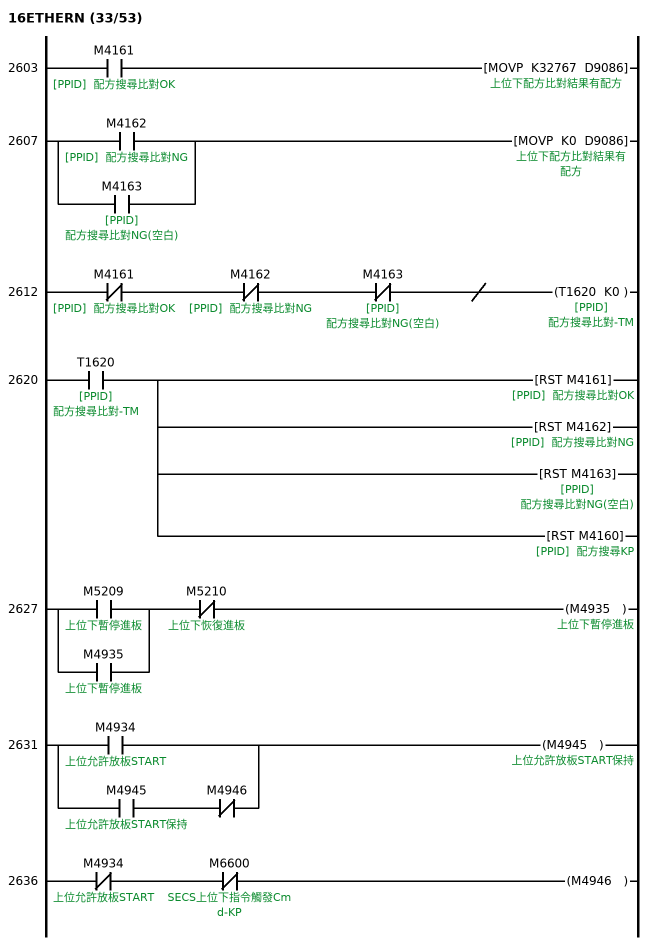
[picture p120: ladder of 16ETHERN, rungs at steps 2603 to 2636]
2603  LD      M4161  ; [PPID]  配方搜尋比對OK
      MOVP    K32767 D9086
2607  LD      M4162  ; [PPID]  配方搜尋比對NG
      OR      M4163  ; [PPID]  配方搜尋比對NG(空白)
      MOVP    K0 D9086
2612  LDI     M4161  ; [PPID]  配方搜尋比對OK
      ANI     M4162  ; [PPID]  配方搜尋比對NG
      ANI     M4163  ; [PPID]  配方搜尋比對NG(空白)
      INV
      OUT     T1620 K0  ; [PPID]  配方搜尋比對-TM
2620  LD      T1620  ; [PPID]  配方搜尋比對-TM
      RST     M4161  ; [PPID]  配方搜尋比對OK
      RST     M4162  ; [PPID]  配方搜尋比對NG
      RST     M4163  ; [PPID]  配方搜尋比對NG(空白)
      RST     M4160  ; [PPID]  配方搜尋KP
2627  LD      M5209  ; 上位下暫停進板
      OR      M4935  ; 上位下暫停進板
      ANI     M5210  ; 上位下恢復進板
      OUT     M4935  ; 上位下暫停進板
2631  LD      M4934  ; 上位允許放板START
      LD      M4945  ; 上位允許放板START保持
      ANI     M4946
      ORB
      OUT     M4945  ; 上位允許放板START保持
2636  LDI     M4934  ; 上位允許放板START
      ANI     M6600  ; SECS上位下指令觸發Cmd-KP
      OUT     M4946
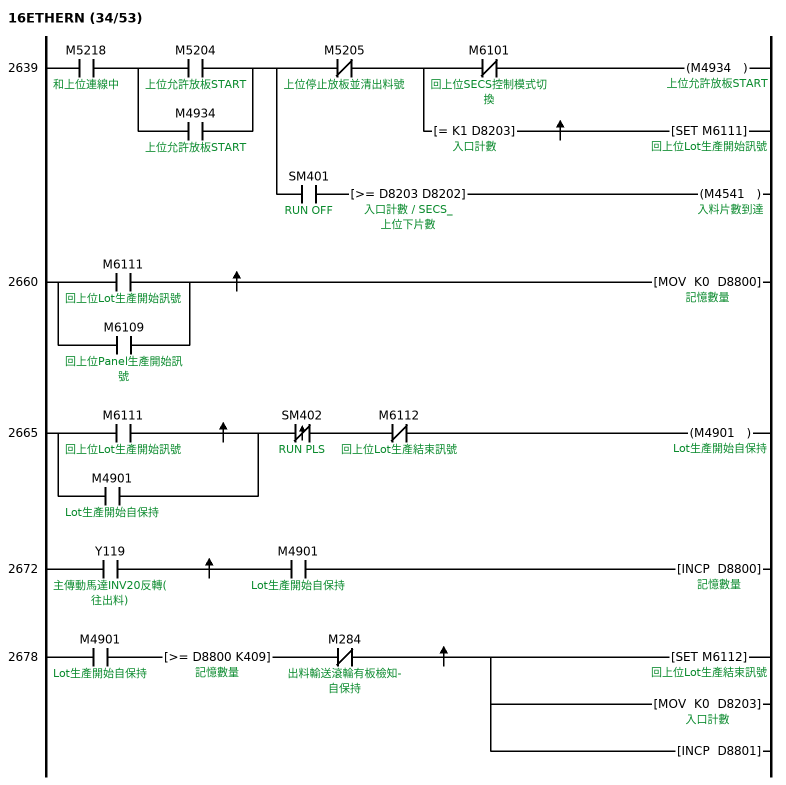
2639  LD      M5218  ; 和上位連線中
      LD      M5204  ; 上位允許放板START
      OR      M4934  ; 上位允許放板START
      ANB
      MPS
      ANI     M5205  ; 上位停止放板並清出料號
      MPS
      ANI     M6101  ; 回上位SECS控制模式切換
      OUT     M4934  ; 上位允許放板START
      MPP
      AND=    K1 D8203  ; 入口計數
      MEP
      SET     M6111  ; 回上位Lot生產開始訊號
      MPP
      AND     SM401  ; RUN OFF
      AND>=   D8203 D8202  ; 入口計數 / SECS_上位下片數
      OUT     M4541  ; 入料片數到達
2660  LD      M6111  ; 回上位Lot生產開始訊號
      OR      M6109  ; 回上位Panel生產開始訊號
      MEP
      MOV     K0 D8800  ; 記憶數量
2665  LD      M6111  ; 回上位Lot生產開始訊號
      MEP
      OR      M4901  ; Lot生產開始自保持
      ANDPI   SM402  ; RUN PLS
      ANI     M6112  ; 回上位Lot生產結束訊號
      OUT     M4901  ; Lot生產開始自保持
2672  LD      Y119  ; 主傳動馬達INV20反轉(往出料)
      MEP
      AND     M4901  ; Lot生產開始自保持
      INCP    D8800
2678  LD      M4901  ; Lot生產開始自保持
      AND>=   D8800 K409  ; 記憶數量
      ANI     M284  ; 出料輸送滾輪有板檢知-自保持
      MEP
      SET     M6112  ; 回上位Lot生產結束訊號
      MOV     K0 D8203
      INCP    D8801
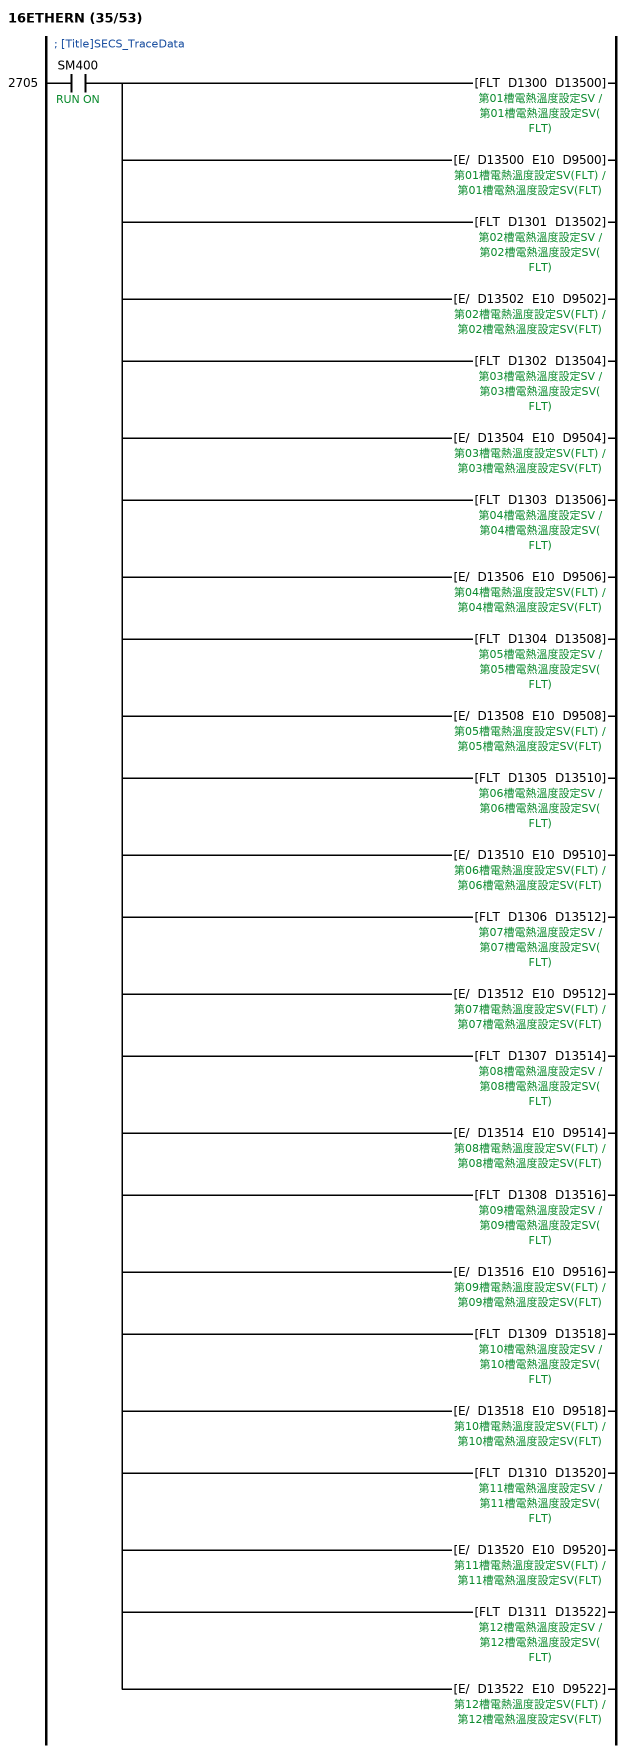
; [Title]SECS_TraceData
2705  LD      SM400  ; RUN ON
      FLT     D1300 D13500  ; 第01槽電熱溫度設定SV / 第01槽電熱溫度設定SV(FLT)
      E/      D13500 E10 D9500  ; 第01槽電熱溫度設定SV(FLT)
      FLT     D1301 D13502  ; 第02槽電熱溫度設定SV / 第02槽電熱溫度設定SV(FLT)
      E/      D13502 E10 D9502  ; 第02槽電熱溫度設定SV(FLT)
      FLT     D1302 D13504  ; 第03槽電熱溫度設定SV / 第03槽電熱溫度設定SV(FLT)
      E/      D13504 E10 D9504  ; 第03槽電熱溫度設定SV(FLT)
      FLT     D1303 D13506  ; 第04槽電熱溫度設定SV / 第04槽電熱溫度設定SV(FLT)
      E/      D13506 E10 D9506  ; 第04槽電熱溫度設定SV(FLT)
      FLT     D1304 D13508  ; 第05槽電熱溫度設定SV / 第05槽電熱溫度設定SV(FLT)
      E/      D13508 E10 D9508  ; 第05槽電熱溫度設定SV(FLT)
      FLT     D1305 D13510  ; 第06槽電熱溫度設定SV / 第06槽電熱溫度設定SV(FLT)
      E/      D13510 E10 D9510  ; 第06槽電熱溫度設定SV(FLT)
      FLT     D1306 D13512  ; 第07槽電熱溫度設定SV / 第07槽電熱溫度設定SV(FLT)
      E/      D13512 E10 D9512  ; 第07槽電熱溫度設定SV(FLT)
      FLT     D1307 D13514  ; 第08槽電熱溫度設定SV / 第08槽電熱溫度設定SV(FLT)
      E/      D13514 E10 D9514  ; 第08槽電熱溫度設定SV(FLT)
      FLT     D1308 D13516  ; 第09槽電熱溫度設定SV / 第09槽電熱溫度設定SV(FLT)
      E/      D13516 E10 D9516  ; 第09槽電熱溫度設定SV(FLT)
      FLT     D1309 D13518  ; 第10槽電熱溫度設定SV / 第10槽電熱溫度設定SV(FLT)
      E/      D13518 E10 D9518  ; 第10槽電熱溫度設定SV(FLT)
      FLT     D1310 D13520  ; 第11槽電熱溫度設定SV / 第11槽電熱溫度設定SV(FLT)
      E/      D13520 E10 D9520  ; 第11槽電熱溫度設定SV(FLT)
      FLT     D1311 D13522  ; 第12槽電熱溫度設定SV / 第12槽電熱溫度設定SV(FLT)
      E/      D13522 E10 D9522  ; 第12槽電熱溫度設定SV(FLT)
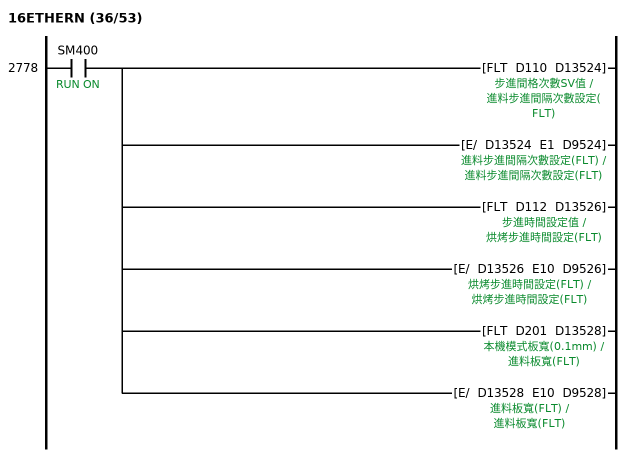
2778  LD      SM400  ; RUN ON
      FLT     D110 D13524  ; 步進間格次數SV值 / 進料步進間隔次數設定(FLT)
      E/      D13524 E1 D9524  ; 進料步進間隔次數設定(FLT)
      FLT     D112 D13526  ; 步進時間設定值 / 烘烤步進時間設定(FLT)
      E/      D13526 E10 D9526  ; 烘烤步進時間設定(FLT)
      FLT     D201 D13528  ; 進料板寬(FLT)
      E/      D13528 E10 D9528  ; 進料板寬(FLT)
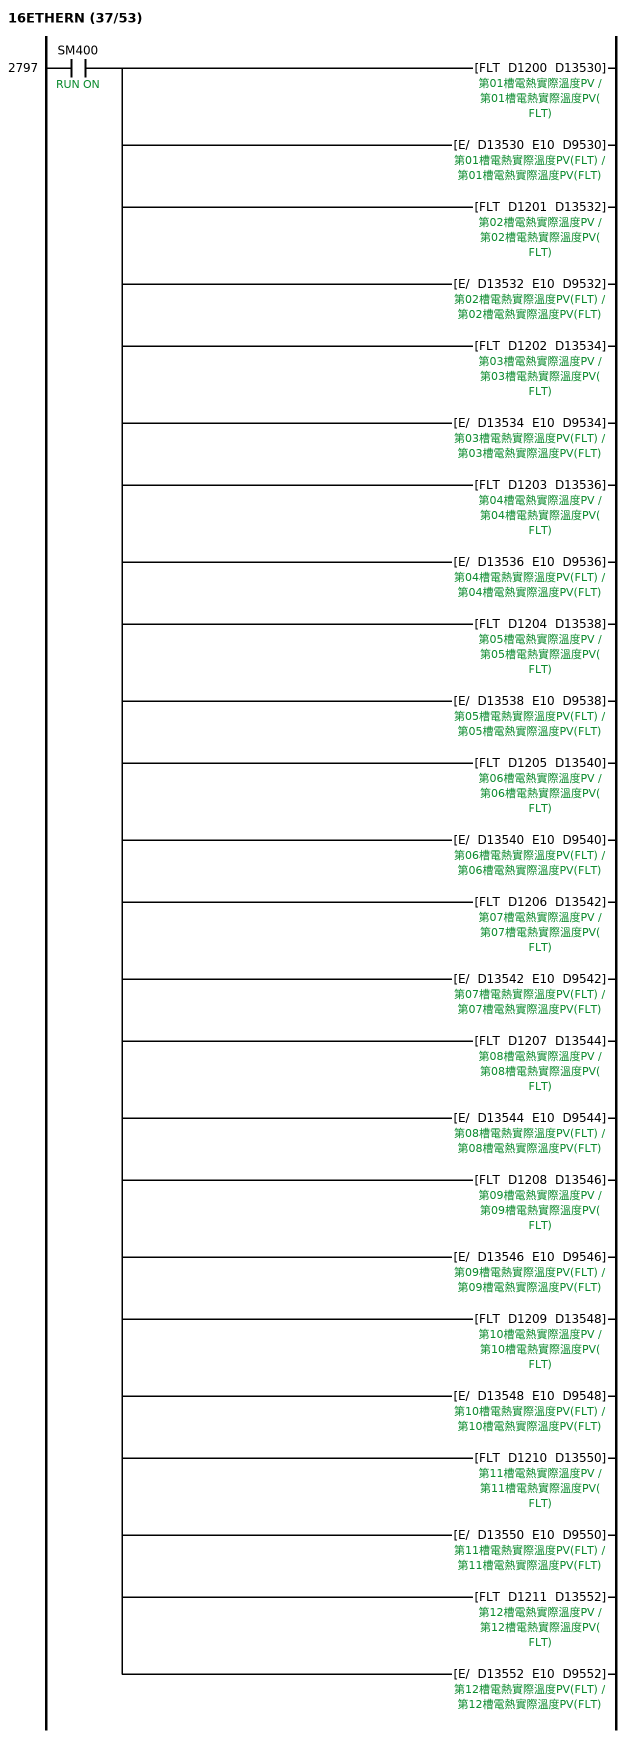
2797  LD      SM400  ; RUN ON
      FLT     D1200 D13530  ; 第01槽電熱實際溫度PV(FLT)
      E/      D13530 E10 D9530  ; 第01槽電熱實際溫度PV(FLT)
      FLT     D1201 D13532  ; 第02槽電熱實際溫度PV(FLT)
      E/      D13532 E10 D9532  ; 第02槽電熱實際溫度PV(FLT)
      FLT     D1202 D13534  ; 第03槽電熱實際溫度PV(FLT)
      E/      D13534 E10 D9534  ; 第03槽電熱實際溫度PV(FLT)
      FLT     D1203 D13536  ; 第04槽電熱實際溫度PV(FLT)
      E/      D13536 E10 D9536  ; 第04槽電熱實際溫度PV(FLT)
      FLT     D1204 D13538  ; 第05槽電熱實際溫度PV(FLT)
      E/      D13538 E10 D9538  ; 第05槽電熱實際溫度PV(FLT)
      FLT     D1205 D13540  ; 第06槽電熱實際溫度PV(FLT)
      E/      D13540 E10 D9540  ; 第06槽電熱實際溫度PV(FLT)
      FLT     D1206 D13542  ; 第07槽電熱實際溫度PV(FLT)
      E/      D13542 E10 D9542  ; 第07槽電熱實際溫度PV(FLT)
      FLT     D1207 D13544  ; 第08槽電熱實際溫度PV(FLT)
      E/      D13544 E10 D9544  ; 第08槽電熱實際溫度PV(FLT)
      FLT     D1208 D13546  ; 第09槽電熱實際溫度PV(FLT)
      E/      D13546 E10 D9546  ; 第09槽電熱實際溫度PV(FLT)
      FLT     D1209 D13548  ; 第10槽電熱實際溫度PV(FLT)
      E/      D13548 E10 D9548  ; 第10槽電熱實際溫度PV(FLT)
      FLT     D1210 D13550  ; 第11槽電熱實際溫度PV(FLT)
      E/      D13550 E10 D9550  ; 第11槽電熱實際溫度PV(FLT)
      FLT     D1211 D13552  ; 第12槽電熱實際溫度PV(FLT)
      E/      D13552 E10 D9552  ; 第12槽電熱實際溫度PV(FLT)
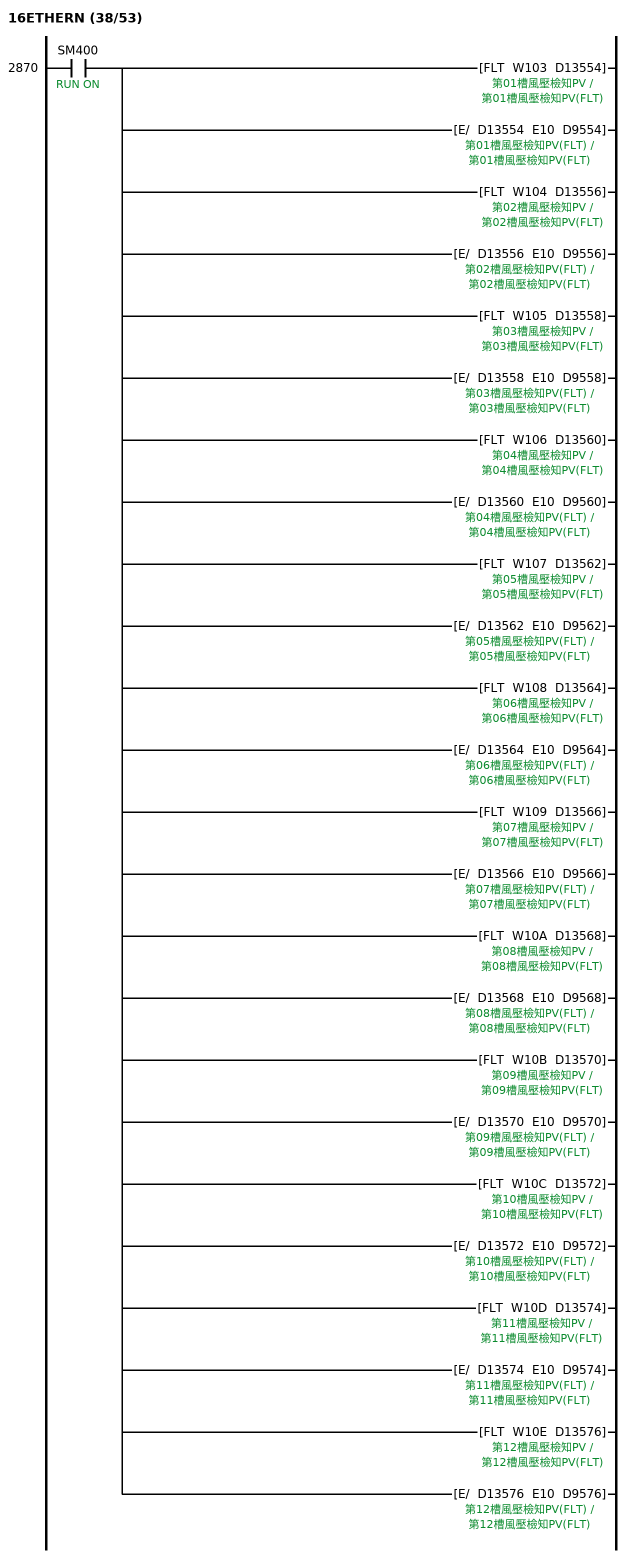
2870  LD      SM400  ; RUN ON
      FLT     W103 D13554  ; 第01槽風壓檢知PV / 第01槽風壓檢知PV(FLT)
      E/      D13554 E10 D9554  ; 第01槽風壓檢知PV(FLT)
      FLT     W104 D13556  ; 第02槽風壓檢知PV / 第02槽風壓檢知PV(FLT)
      E/      D13556 E10 D9556  ; 第02槽風壓檢知PV(FLT)
      FLT     W105 D13558  ; 第03槽風壓檢知PV / 第03槽風壓檢知PV(FLT)
      E/      D13558 E10 D9558  ; 第03槽風壓檢知PV(FLT)
      FLT     W106 D13560  ; 第04槽風壓檢知PV / 第04槽風壓檢知PV(FLT)
      E/      D13560 E10 D9560  ; 第04槽風壓檢知PV(FLT)
      FLT     W107 D13562  ; 第05槽風壓檢知PV / 第05槽風壓檢知PV(FLT)
      E/      D13562 E10 D9562  ; 第05槽風壓檢知PV(FLT)
      FLT     W108 D13564  ; 第06槽風壓檢知PV / 第06槽風壓檢知PV(FLT)
      E/      D13564 E10 D9564  ; 第06槽風壓檢知PV(FLT)
      FLT     W109 D13566  ; 第07槽風壓檢知PV / 第07槽風壓檢知PV(FLT)
      E/      D13566 E10 D9566  ; 第07槽風壓檢知PV(FLT)
      FLT     W10A D13568  ; 第08槽風壓檢知PV / 第08槽風壓檢知PV(FLT)
      E/      D13568 E10 D9568  ; 第08槽風壓檢知PV(FLT)
      FLT     W10B D13570  ; 第09槽風壓檢知PV / 第09槽風壓檢知PV(FLT)
      E/      D13570 E10 D9570  ; 第09槽風壓檢知PV(FLT)
      FLT     W10C D13572  ; 第10槽風壓檢知PV / 第10槽風壓檢知PV(FLT)
      E/      D13572 E10 D9572  ; 第10槽風壓檢知PV(FLT)
      FLT     W10D D13574  ; 第11槽風壓檢知PV / 第11槽風壓檢知PV(FLT)
      E/      D13574 E10 D9574  ; 第11槽風壓檢知PV(FLT)
      FLT     W10E D13576  ; 第12槽風壓檢知PV / 第12槽風壓檢知PV(FLT)
      E/      D13576 E10 D9576  ; 第12槽風壓檢知PV(FLT)
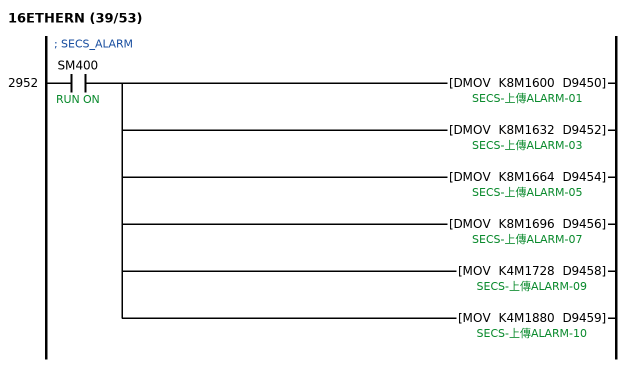
; SECS_ALARM
2952  LD      SM400  ; RUN ON
      DMOV    K8M1600 D9450  ; SECS-上傳ALARM-01
      DMOV    K8M1632 D9452  ; SECS-上傳ALARM-03
      DMOV    K8M1664 D9454  ; 出料風車1過載異常 / SECS-上傳ALARM-05
      DMOV    K8M1696 D9456  ; 進料夾爪開異常 / SECS-上傳ALARM-07
      MOV     K4M1728 D9458  ; 緊急停止異常 / SECS-上傳ALARM-09
      MOV     K4M1880 D9459  ; #01分路開關跳脫 / SECS-上傳ALARM-10
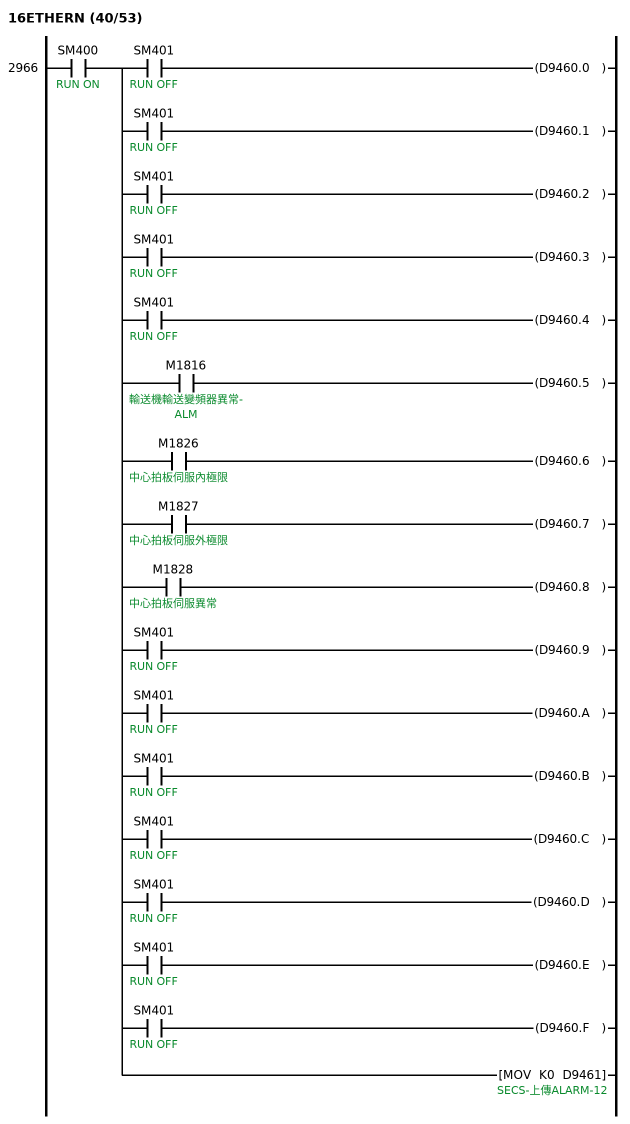
2966  LD      SM400  ; RUN ON
      MPS
      AND     SM401  ; RUN OFF
      OUT     D9460.0
      MRD
      AND     SM401  ; RUN OFF
      OUT     D9460.1
      MRD
      AND     SM401  ; RUN OFF
      OUT     D9460.2
      MRD
      AND     SM401  ; RUN OFF
      OUT     D9460.3
      MRD
      AND     SM401  ; RUN OFF
      OUT     D9460.4
      MRD
      AND     M1816  ; 輸送機輸送變頻器異常-ALM
      OUT     D9460.5
      MRD
      AND     M1826  ; 中心拍板伺服內極限
      OUT     D9460.6
      MRD
      AND     M1827  ; 中心拍板伺服外極限
      OUT     D9460.7
      MRD
      AND     M1828  ; 中心拍板伺服異常
      OUT     D9460.8
      MRD
      AND     SM401  ; RUN OFF
      OUT     D9460.9
      MRD
      AND     SM401  ; RUN OFF
      OUT     D9460.A
      MRD
      AND     SM401  ; RUN OFF
      OUT     D9460.B
      MRD
      AND     SM401  ; RUN OFF
      OUT     D9460.C
      MRD
      AND     SM401  ; RUN OFF
      OUT     D9460.D
      MRD
      AND     SM401  ; RUN OFF
      OUT     D9460.E
      MRD
      AND     SM401  ; RUN OFF
      OUT     D9460.F
      MPP
      MOV     K0 D9461  ; SECS-上傳ALARM-12
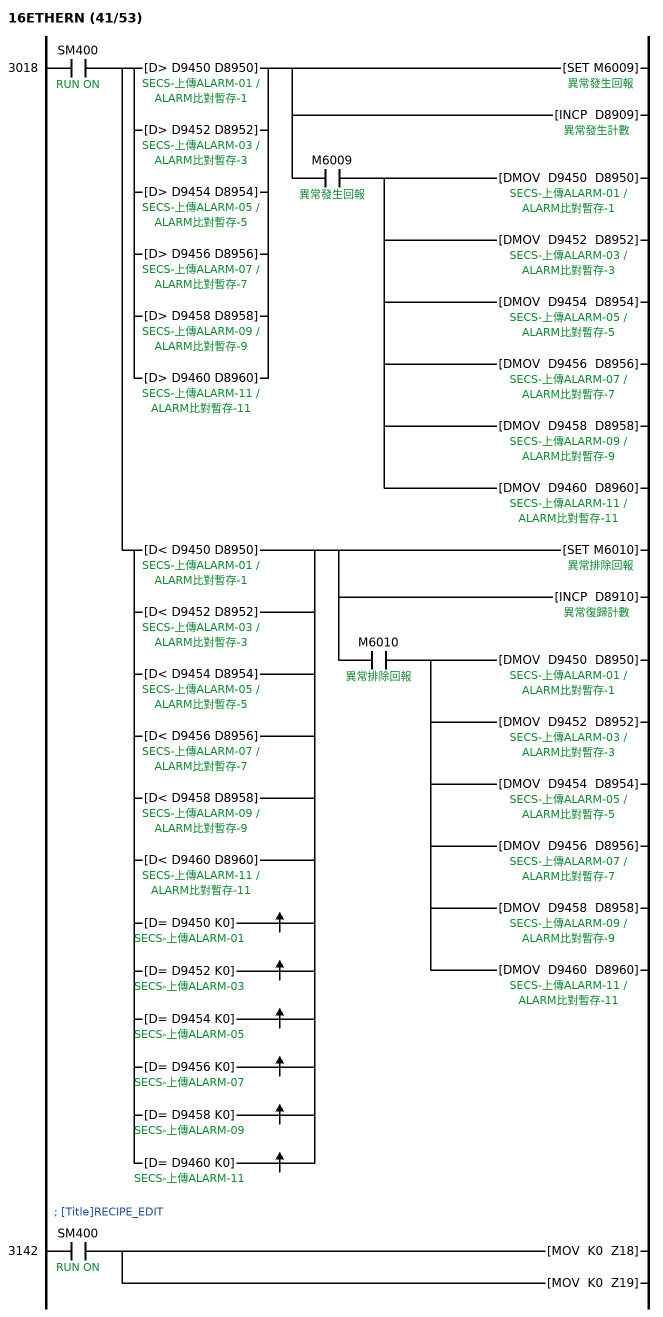
3018  LD      SM400  ; RUN ON
      MPS
      LDD>    D9450 D8950  ; SECS-上傳ALARM-01 / ALARM比對暫存-1
      ORD>    D9452 D8952  ; SECS-上傳ALARM-03 / ALARM比對暫存-3
      ORD>    D9454 D8954  ; SECS-上傳ALARM-05 / ALARM比對暫存-5
      ORD>    D9456 D8956  ; SECS-上傳ALARM-07 / ALARM比對暫存-7
      ORD>    D9458 D8958  ; SECS-上傳ALARM-09 / ALARM比對暫存-9
      ORD>    D9460 D8960  ; SECS-上傳ALARM-11 / ALARM比對暫存-11
      ANB
      SET     M6009  ; 異常發生回報
      INCP    D8909  ; 異常發生計數
      AND     M6009  ; 異常發生回報
      DMOV    D9450 D8950
      DMOV    D9452 D8952
      DMOV    D9454 D8954
      DMOV    D9456 D8956
      DMOV    D9458 D8958
      DMOV    D9460 D8960
      MPP
      LDD<    D9450 D8950  ; SECS-上傳ALARM-01 / ALARM比對暫存-1
      ORD<    D9452 D8952  ; SECS-上傳ALARM-03 / ALARM比對暫存-3
      ORD<    D9454 D8954  ; SECS-上傳ALARM-05 / ALARM比對暫存-5
      ORD<    D9456 D8956  ; SECS-上傳ALARM-07 / ALARM比對暫存-7
      ORD<    D9458 D8958  ; SECS-上傳ALARM-09 / ALARM比對暫存-9
      ORD<    D9460 D8960  ; SECS-上傳ALARM-11 / ALARM比對暫存-11
      LDD=    D9450 K0  ; SECS-上傳ALARM-01
      MEP
      ORB
      LDD=    D9452 K0  ; SECS-上傳ALARM-03
      MEP
      ORB
      LDD=    D9454 K0  ; SECS-上傳ALARM-05
      MEP
      ORB
      LDD=    D9456 K0  ; SECS-上傳ALARM-07
      MEP
      ORB
      LDD=    D9458 K0  ; SECS-上傳ALARM-09
      MEP
      ORB
      LDD=    D9460 K0  ; SECS-上傳ALARM-11
      MEP
      ORB
      ANB
      SET     M6010  ; 異常排除回報
      INCP    D8910  ; 異常復歸計數
      AND     M6010  ; 異常排除回報
      DMOV    D9450 D8950
      DMOV    D9452 D8952
      DMOV    D9454 D8954
      DMOV    D9456 D8956
      DMOV    D9458 D8958
      DMOV    D9460 D8960
; [Title]RECIPE_EDIT
3142  LD      SM400  ; RUN ON
      MOV     K0 Z18
      MOV     K0 Z19
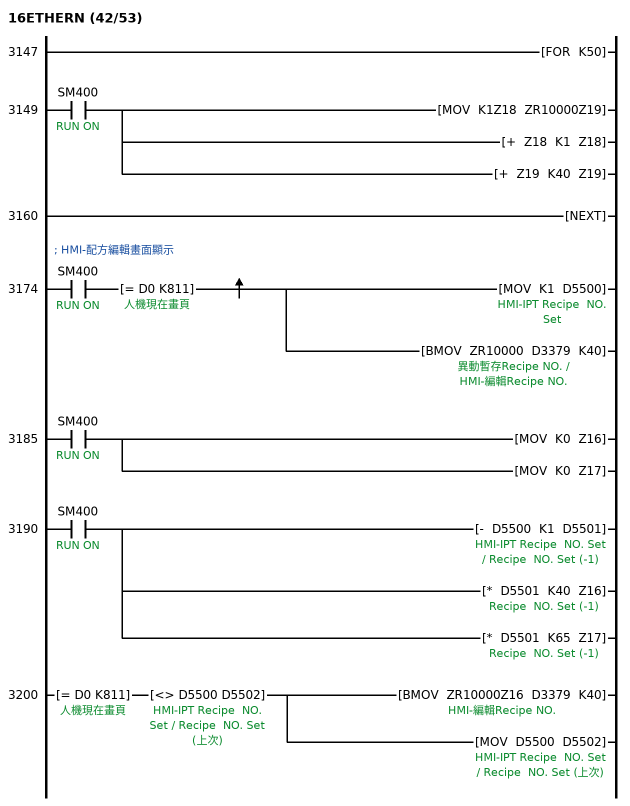
3147  FOR     K50
3149  LD      SM400  ; RUN ON
      MOV     K1Z18 ZR10000Z19
      +       Z18 K1 Z18
      +       Z19 K40 Z19
3160  NEXT
; HMI-配方編輯畫面顯示
3174  LD      SM400  ; RUN ON
      AND=    D0 K811  ; 人機現在畫頁
      MEP
      MOV     K1 D5500  ; HMI-IPT Recipe  NO. Set
      BMOV    ZR10000 D3379 K40  ; 異動暫存Recipe NO. / HMI-編輯Recipe NO.
3185  LD      SM400  ; RUN ON
      MOV     K0 Z16
      MOV     K0 Z17
3190  LD      SM400  ; RUN ON
      -       D5500 K1 D5501  ; Recipe  NO. Set (-1)
      *       D5501 K40 Z16
      *       D5501 K65 Z17
3200  LD=     D0 K811  ; 人機現在畫頁
      AND<>   D5500 D5502  ; HMI-IPT Recipe  NO. Set / Recipe  NO. Set (上次)
      BMOV    ZR10000Z16 D3379 K40
      MOV     D5500 D5502
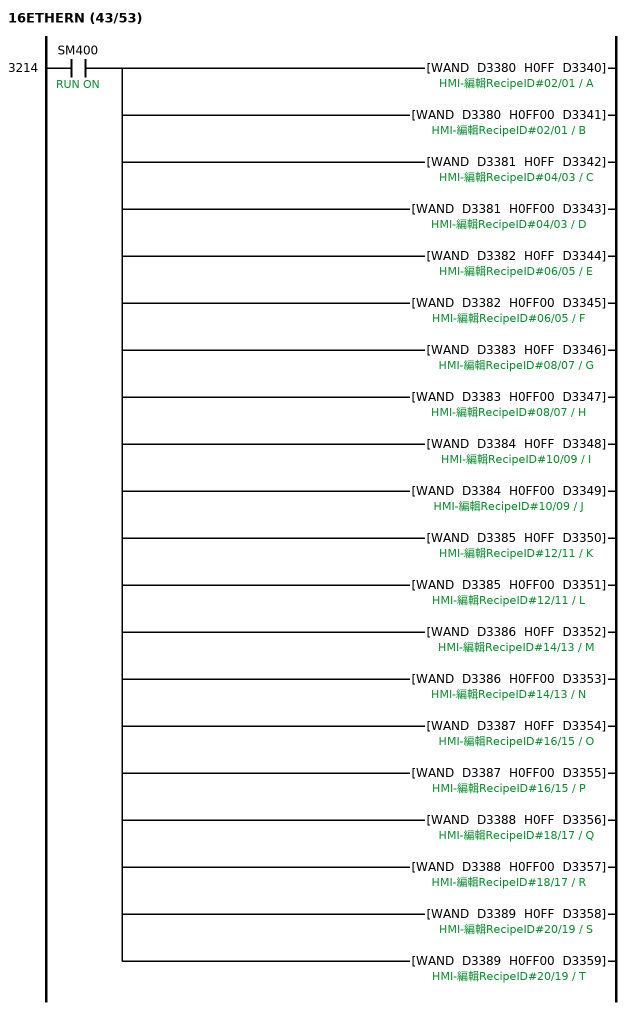
3214  LD      SM400  ; RUN ON
      WAND    D3380 H0FF D3340  ; HMI-編輯RecipeID#02/01 / A
      WAND    D3380 H0FF00 D3341  ; B
      WAND    D3381 H0FF D3342  ; HMI-編輯RecipeID#04/03 / C
      WAND    D3381 H0FF00 D3343  ; D
      WAND    D3382 H0FF D3344  ; HMI-編輯RecipeID#06/05 / E
      WAND    D3382 H0FF00 D3345  ; F
      WAND    D3383 H0FF D3346  ; HMI-編輯RecipeID#08/07 / G
      WAND    D3383 H0FF00 D3347  ; H
      WAND    D3384 H0FF D3348  ; HMI-編輯RecipeID#10/09 / I
      WAND    D3384 H0FF00 D3349  ; J
      WAND    D3385 H0FF D3350  ; HMI-編輯RecipeID#12/11 / K
      WAND    D3385 H0FF00 D3351  ; L
      WAND    D3386 H0FF D3352  ; HMI-編輯RecipeID#14/13 / M
      WAND    D3386 H0FF00 D3353  ; N
      WAND    D3387 H0FF D3354  ; HMI-編輯RecipeID#16/15 / O
      WAND    D3387 H0FF00 D3355  ; P
      WAND    D3388 H0FF D3356  ; HMI-編輯RecipeID#18/17 / Q
      WAND    D3388 H0FF00 D3357  ; R
      WAND    D3389 H0FF D3358  ; HMI-編輯RecipeID#20/19 / S
      WAND    D3389 H0FF00 D3359  ; T
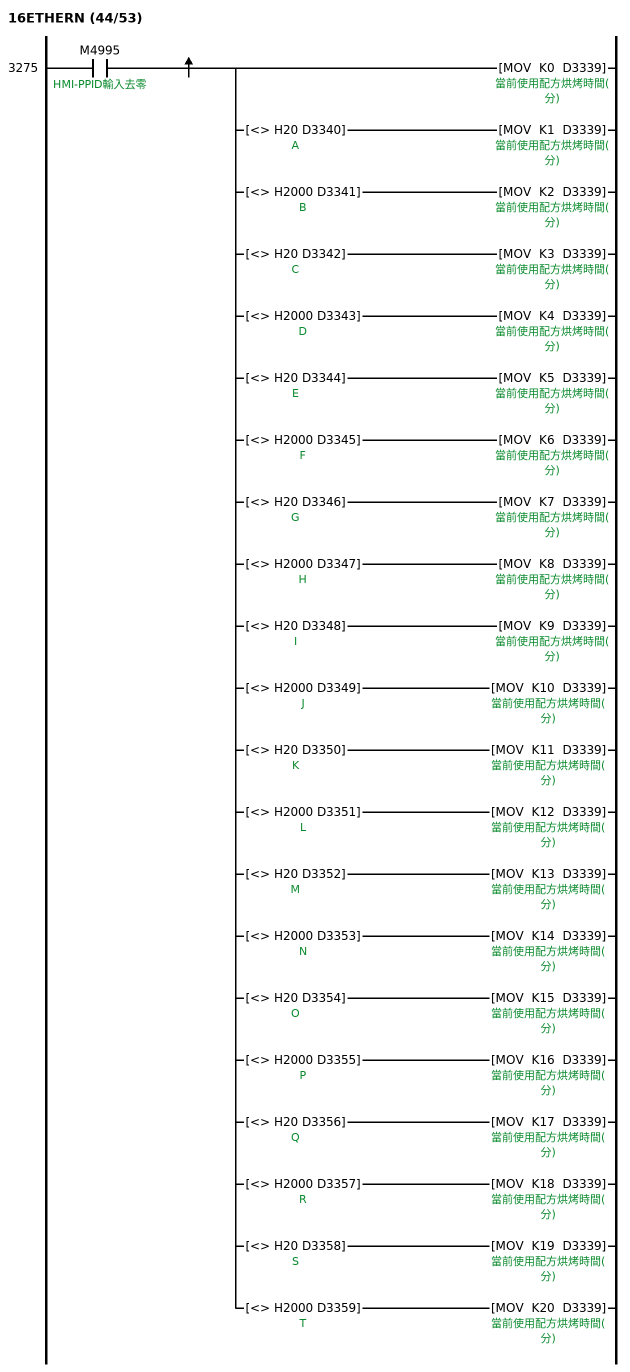
3275  LD      M4995  ; HMI-PPID輸入去零
      MEP
      MOV     K0 D3339  ; 當前使用配方烘烤時間(分)
      MPS
      AND<>   H20 D3340  ; A
      MOV     K1 D3339
      MRD
      AND<>   H2000 D3341  ; B
      MOV     K2 D3339
      MRD
      AND<>   H20 D3342  ; C
      MOV     K3 D3339
      MRD
      AND<>   H2000 D3343  ; D
      MOV     K4 D3339
      MRD
      AND<>   H20 D3344  ; E
      MOV     K5 D3339
      MRD
      AND<>   H2000 D3345  ; F
      MOV     K6 D3339
      MRD
      AND<>   H20 D3346  ; G
      MOV     K7 D3339
      MRD
      AND<>   H2000 D3347  ; H
      MOV     K8 D3339
      MRD
      AND<>   H20 D3348  ; I
      MOV     K9 D3339
      MRD
      AND<>   H2000 D3349  ; J
      MOV     K10 D3339
      MRD
      AND<>   H20 D3350  ; K
      MOV     K11 D3339
      MRD
      AND<>   H2000 D3351  ; L
      MOV     K12 D3339
      MRD
      AND<>   H20 D3352  ; M
      MOV     K13 D3339
      MRD
      AND<>   H2000 D3353  ; N
      MOV     K14 D3339
      MRD
      AND<>   H20 D3354  ; O
      MOV     K15 D3339
      MRD
      AND<>   H2000 D3355  ; P
      MOV     K16 D3339
      MRD
      AND<>   H20 D3356  ; Q
      MOV     K17 D3339
      MRD
      AND<>   H2000 D3357  ; R
      MOV     K18 D3339
      MRD
      AND<>   H20 D3358  ; S
      MOV     K19 D3339
      MPP
      AND<>   H2000 D3359  ; T
      MOV     K20 D3339
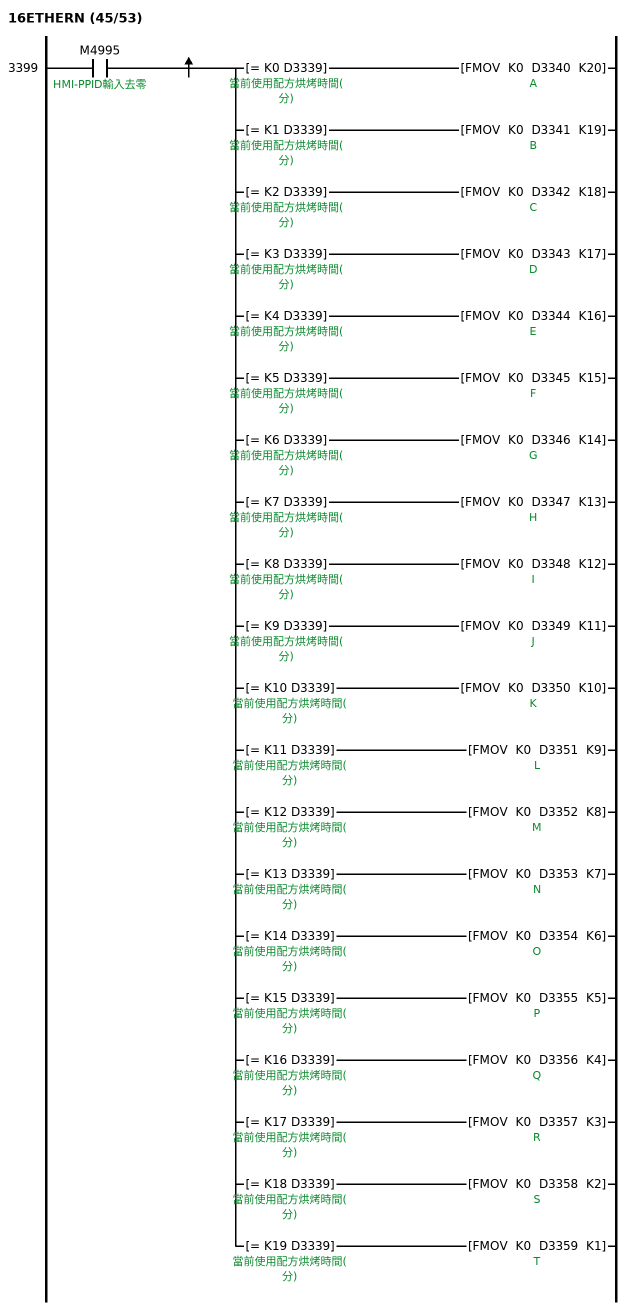
3399  LD      M4995  ; HMI-PPID輸入去零
      MEP
      MPS
      AND=    K0 D3339  ; 當前使用配方烘烤時間(分)
      FMOV    K0 D3340 K20
      MRD
      AND=    K1 D3339  ; 當前使用配方烘烤時間(分)
      FMOV    K0 D3341 K19
      MRD
      AND=    K2 D3339  ; 當前使用配方烘烤時間(分)
      FMOV    K0 D3342 K18
      MRD
      AND=    K3 D3339  ; 當前使用配方烘烤時間(分)
      FMOV    K0 D3343 K17
      MRD
      AND=    K4 D3339  ; 當前使用配方烘烤時間(分)
      FMOV    K0 D3344 K16
      MRD
      AND=    K5 D3339  ; 當前使用配方烘烤時間(分)
      FMOV    K0 D3345 K15
      MRD
      AND=    K6 D3339  ; 當前使用配方烘烤時間(分)
      FMOV    K0 D3346 K14
      MRD
      AND=    K7 D3339  ; 當前使用配方烘烤時間(分)
      FMOV    K0 D3347 K13
      MRD
      AND=    K8 D3339  ; 當前使用配方烘烤時間(分)
      FMOV    K0 D3348 K12
      MRD
      AND=    K9 D3339  ; 當前使用配方烘烤時間(分)
      FMOV    K0 D3349 K11
      MRD
      AND=    K10 D3339  ; 當前使用配方烘烤時間(分)
      FMOV    K0 D3350 K10
      MRD
      AND=    K11 D3339  ; 當前使用配方烘烤時間(分)
      FMOV    K0 D3351 K9
      MRD
      AND=    K12 D3339  ; 當前使用配方烘烤時間(分)
      FMOV    K0 D3352 K8
      MRD
      AND=    K13 D3339  ; 當前使用配方烘烤時間(分)
      FMOV    K0 D3353 K7
      MRD
      AND=    K14 D3339  ; 當前使用配方烘烤時間(分)
      FMOV    K0 D3354 K6
      MRD
      AND=    K15 D3339  ; 當前使用配方烘烤時間(分)
      FMOV    K0 D3355 K5
      MRD
      AND=    K16 D3339  ; 當前使用配方烘烤時間(分)
      FMOV    K0 D3356 K4
      MRD
      AND=    K17 D3339  ; 當前使用配方烘烤時間(分)
      FMOV    K0 D3357 K3
      MRD
      AND=    K18 D3339  ; 當前使用配方烘烤時間(分)
      FMOV    K0 D3358 K2
      MPP
      AND=    K19 D3339  ; 當前使用配方烘烤時間(分)
      FMOV    K0 D3359 K1
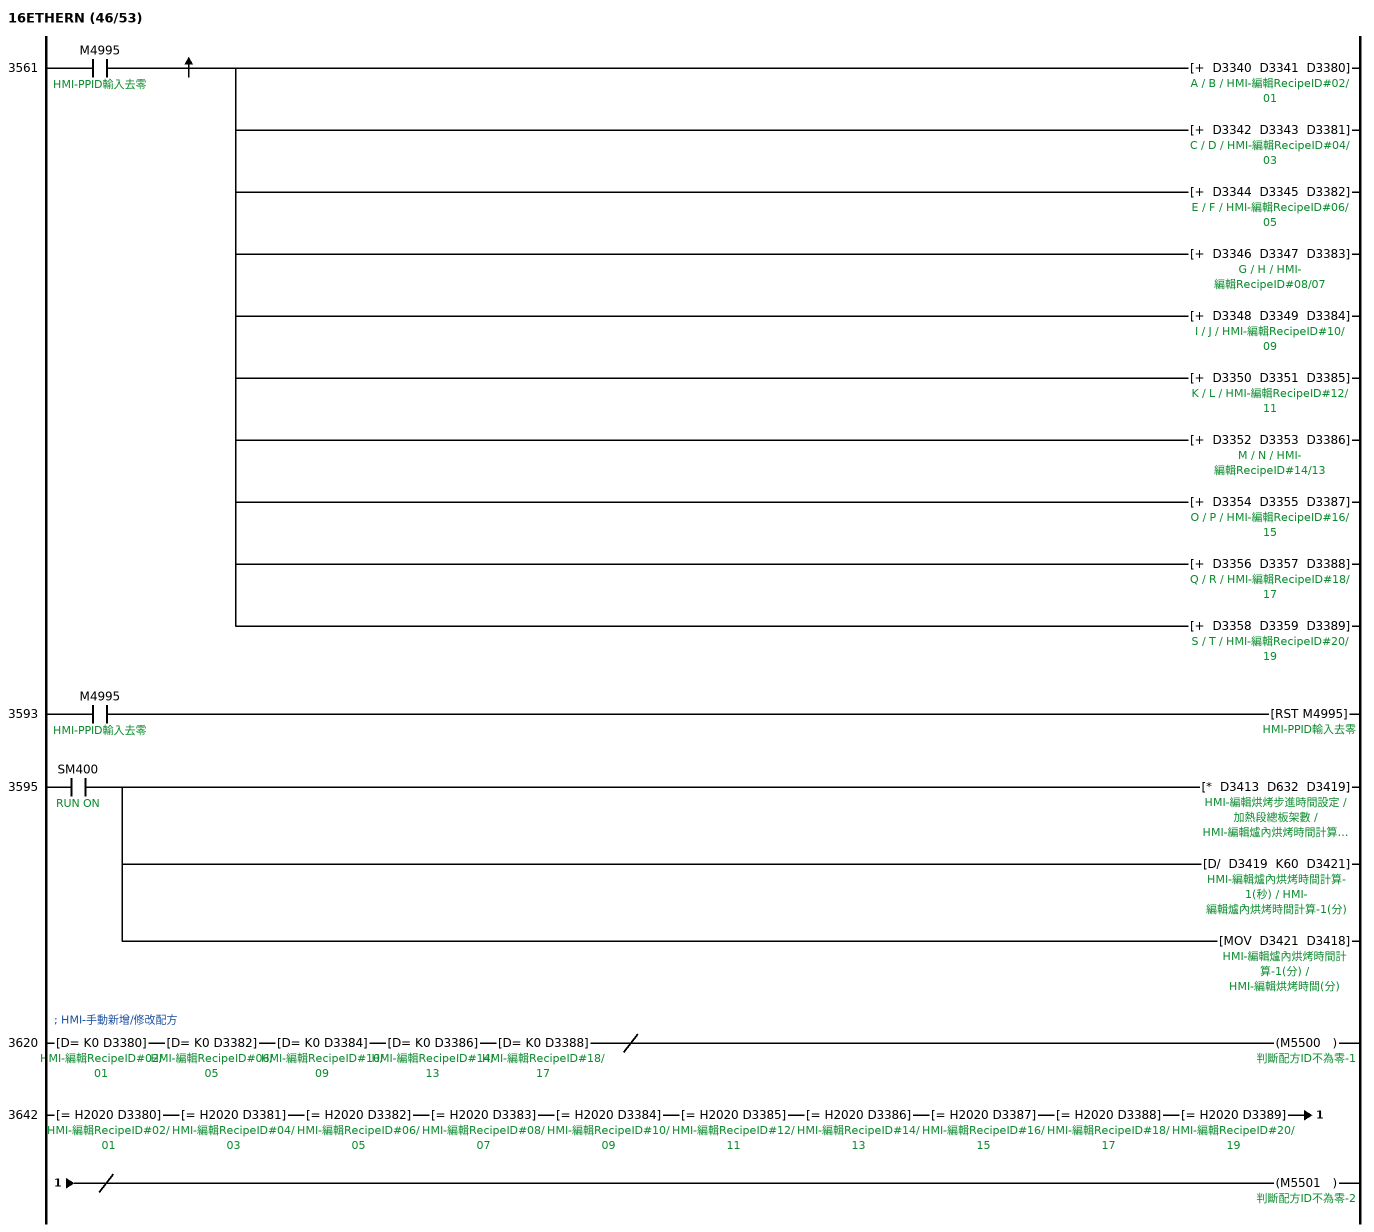
3561  LD      M4995  ; HMI-PPID輸入去零
      MEP
      +       D3340 D3341 D3380
      +       D3342 D3343 D3381
      +       D3344 D3345 D3382
      +       D3346 D3347 D3383
      +       D3348 D3349 D3384
      +       D3350 D3351 D3385
      +       D3352 D3353 D3386
      +       D3354 D3355 D3387
      +       D3356 D3357 D3388
      +       D3358 D3359 D3389
3593  LD      M4995  ; HMI-PPID輸入去零
      RST     M4995  ; HMI-PPID輸入去零
3595  LD      SM400  ; RUN ON
      *       D3413 D632 D3419  ; HMI-編輯烘烤步進時間設定 / 加熱段總板架數 / HMI-編輯爐內烘烤時間計算-1(秒)
      D/      D3419 K60 D3421  ; HMI-編輯爐內烘烤時間計算-1(分)
      MOV     D3421 D3418  ; HMI-編輯烘烤時間(分)
; HMI-手動新增/修改配方
3620  LDD=    K0 D3380  ; HMI-編輯RecipeID#02/01
      ANDD=   K0 D3382  ; HMI-編輯RecipeID#06/05
      ANDD=   K0 D3384  ; HMI-編輯RecipeID#10/09
      ANDD=   K0 D3386  ; HMI-編輯RecipeID#14/13
      ANDD=   K0 D3388  ; HMI-編輯RecipeID#18/17
      INV
      OUT     M5500  ; 判斷配方ID不為零-1
3642  LD=     H2020 D3380  ; HMI-編輯RecipeID#02/01
      AND=    H2020 D3381  ; HMI-編輯RecipeID#04/03
      AND=    H2020 D3382  ; HMI-編輯RecipeID#06/05
      AND=    H2020 D3383  ; HMI-編輯RecipeID#08/07
      AND=    H2020 D3384  ; HMI-編輯RecipeID#10/09
      AND=    H2020 D3385  ; HMI-編輯RecipeID#12/11
      AND=    H2020 D3386  ; HMI-編輯RecipeID#14/13
      AND=    H2020 D3387  ; HMI-編輯RecipeID#16/15
      AND=    H2020 D3388  ; HMI-編輯RecipeID#18/17
      AND=    H2020 D3389  ; HMI-編輯RecipeID#20/19
      INV
      OUT     M5501  ; 判斷配方ID不為零-2
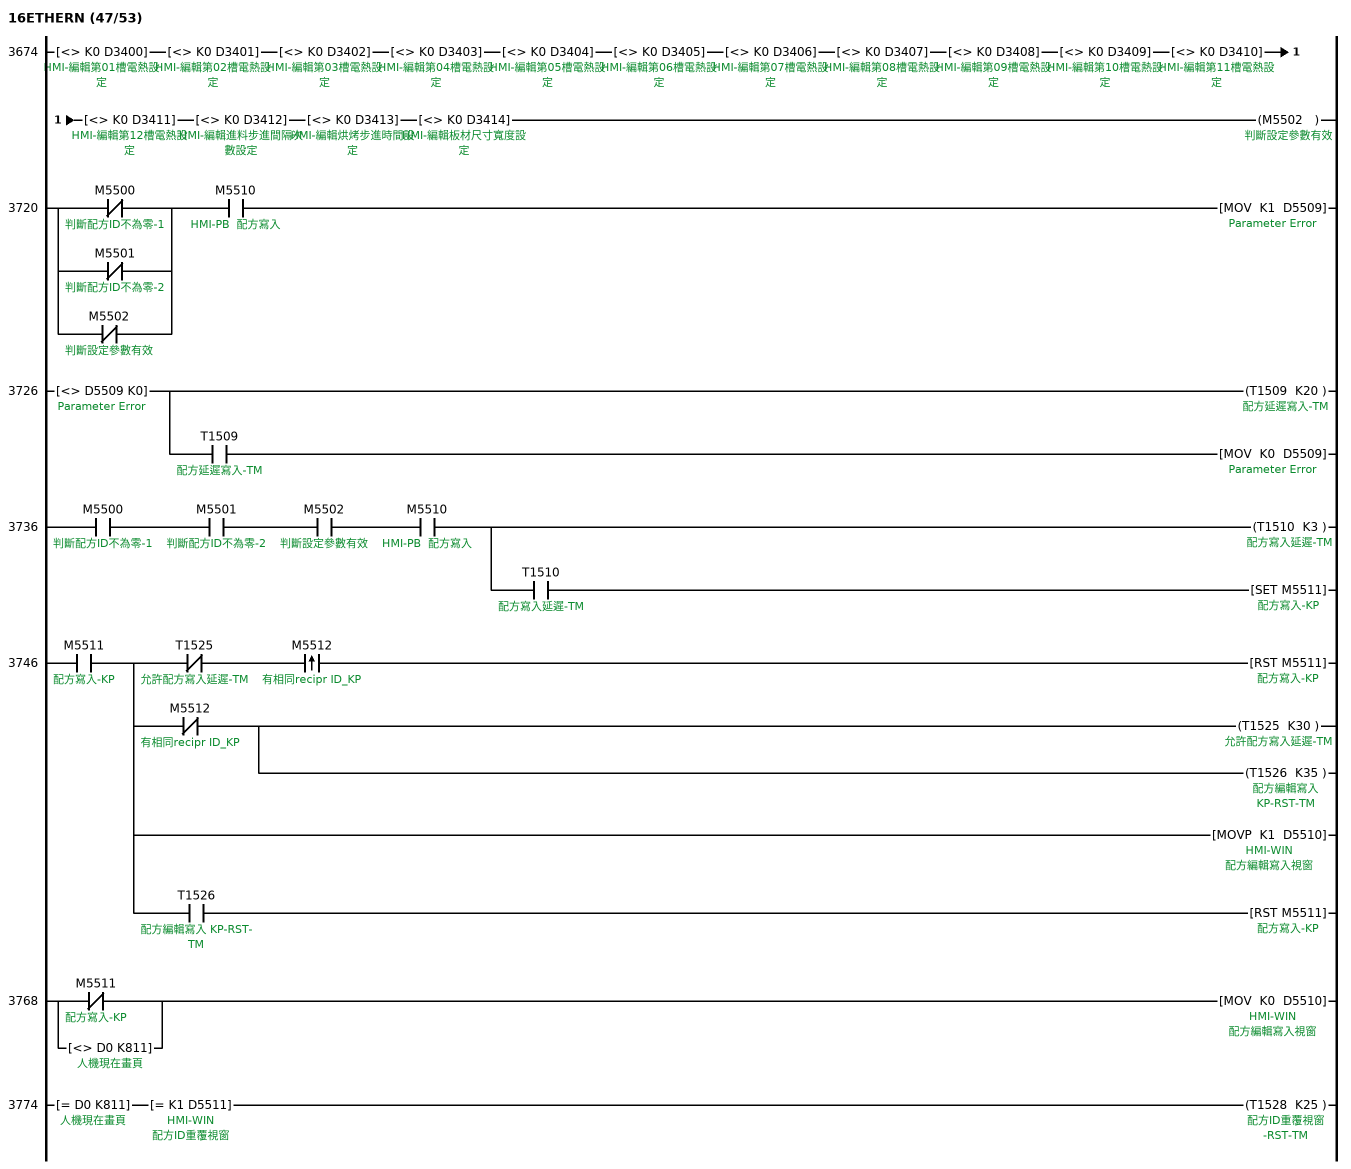
3674  LD<>    K0 D3400  ; HMI-編輯第01槽電熱設定
      AND<>   K0 D3401  ; HMI-編輯第02槽電熱設定
      AND<>   K0 D3402  ; HMI-編輯第03槽電熱設定
      AND<>   K0 D3403  ; HMI-編輯第04槽電熱設定
      AND<>   K0 D3404  ; HMI-編輯第05槽電熱設定
      AND<>   K0 D3405  ; HMI-編輯第06槽電熱設定
      AND<>   K0 D3406  ; HMI-編輯第07槽電熱設定
      AND<>   K0 D3407  ; HMI-編輯第08槽電熱設定
      AND<>   K0 D3408  ; HMI-編輯第09槽電熱設定
      AND<>   K0 D3409  ; HMI-編輯第10槽電熱設定
      AND<>   K0 D3410  ; HMI-編輯第11槽電熱設定
      AND<>   K0 D3411  ; HMI-編輯第12槽電熱設定
      AND<>   K0 D3412  ; HMI-編輯進料步進間隔次數設定
      AND<>   K0 D3413  ; HMI-編輯烘烤步進時間設定
      AND<>   K0 D3414  ; HMI-編輯板材尺寸寬度設定
      OUT     M5502  ; 判斷設定參數有效
3720  LDI     M5500  ; 判斷配方ID不為零-1
      ORI     M5501  ; 判斷配方ID不為零-2
      ORI     M5502  ; 判斷設定參數有效
      AND     M5510  ; HMI-PB  配方寫入
      MOV     K1 D5509  ; Parameter Error
3726  LD<>    D5509 K0  ; Parameter Error
      OUT     T1509 K20  ; 配方延遲寫入-TM
      AND     T1509  ; 配方延遲寫入-TM
      MOV     K0 D5509
3736  LD      M5500  ; 判斷配方ID不為零-1
      AND     M5501  ; 判斷配方ID不為零-2
      AND     M5502  ; 判斷設定參數有效
      AND     M5510  ; HMI-PB  配方寫入
      OUT     T1510 K3  ; 配方寫入延遲-TM
      AND     T1510  ; 配方寫入延遲-TM
      SET     M5511  ; 配方寫入-KP
3746  LD      M5511  ; 配方寫入-KP
      MPS
      ANI     T1525  ; 允許配方寫入延遲-TM
      ANDP    M5512  ; 有相同recipr ID_KP
      RST     M5511  ; 配方寫入-KP
      MRD
      ANI     M5512  ; 有相同recipr ID_KP
      OUT     T1525 K30  ; 允許配方寫入延遲-TM
      OUT     T1526 K35  ; 配方編輯寫入 KP-RST-TM
      MPP
      MOVP    K1 D5510  ; HMI-WIN 配方編輯寫入視窗
      AND     T1526  ; 配方編輯寫入 KP-RST-TM
      RST     M5511  ; 配方寫入-KP
3768  LDI     M5511  ; 配方寫入-KP
      OR<>    D0 K811  ; 人機現在畫頁
      MOV     K0 D5510
3774  LD=     D0 K811  ; 人機現在畫頁
      AND=    K1 D5511  ; HMI-WIN 配方ID重覆視窗
      OUT     T1528 K25  ; 配方ID重覆視窗  -RST-TM
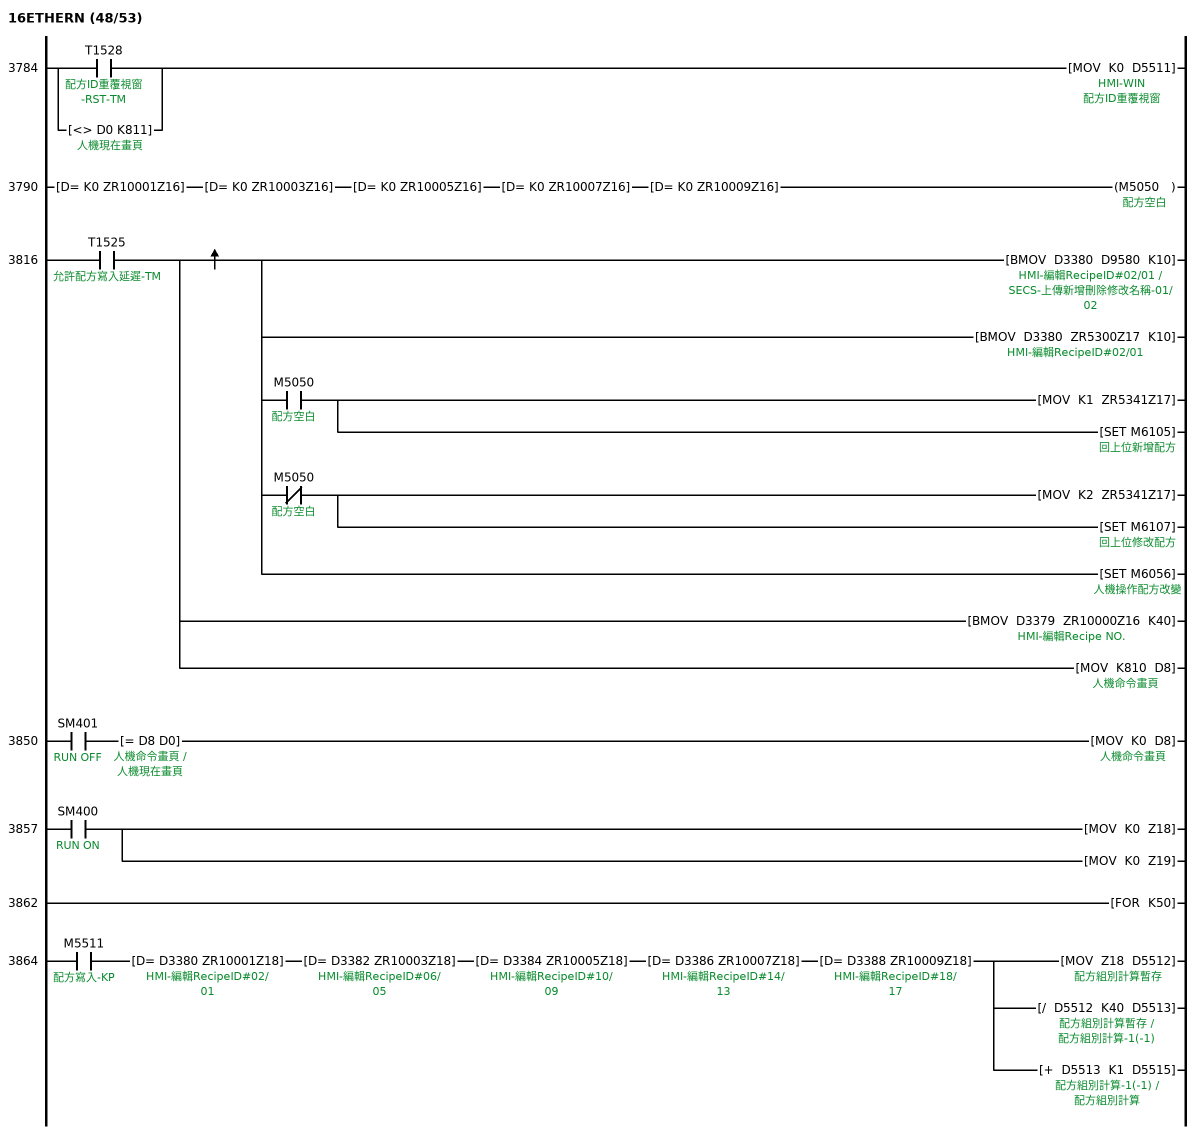
3784  LD      T1528  ; 配方ID重覆視窗  -RST-TM
      OR<>    D0 K811  ; 人機現在畫頁
      MOV     K0 D5511
3790  LDD=    K0 ZR10001Z16
      ANDD=   K0 ZR10003Z16
      ANDD=   K0 ZR10005Z16
      ANDD=   K0 ZR10007Z16
      ANDD=   K0 ZR10009Z16
      OUT     M5050  ; 配方空白
3816  LD      T1525  ; 允許配方寫入延遲-TM
      MPS
      MEP
      BMOV    D3380 D9580 K10  ; SECS-上傳新增刪除修改名稱-01/02
      BMOV    D3380 ZR5300Z17 K10
      MPS
      AND     M5050  ; 配方空白
      MOV     K1 ZR5341Z17
      SET     M6105  ; 回上位新增配方
      MRD
      ANI     M5050  ; 配方空白
      MOV     K2 ZR5341Z17
      SET     M6107  ; 回上位修改配方
      MPP
      SET     M6056  ; 人機操作配方改變
      MPP
      BMOV    D3379 ZR10000Z16 K40
      MOV     K810 D8
3850  LD      SM401  ; RUN OFF
      AND=    D8 D0  ; 人機命令畫頁 / 人機現在畫頁
      MOV     K0 D8
3857  LD      SM400  ; RUN ON
      MOV     K0 Z18
      MOV     K0 Z19
3862  FOR     K50
3864  LD      M5511  ; 配方寫入-KP
      ANDD=   D3380 ZR10001Z18  ; HMI-編輯RecipeID#02/01
      ANDD=   D3382 ZR10003Z18  ; HMI-編輯RecipeID#06/05
      ANDD=   D3384 ZR10005Z18  ; HMI-編輯RecipeID#10/09
      ANDD=   D3386 ZR10007Z18  ; HMI-編輯RecipeID#14/13
      ANDD=   D3388 ZR10009Z18  ; HMI-編輯RecipeID#18/17
      MOV     Z18 D5512  ; 配方組別計算暫存
      /       D5512 K40 D5513  ; 配方組別計算-1(-1)
      +       D5513 K1 D5515  ; 配方組別計算
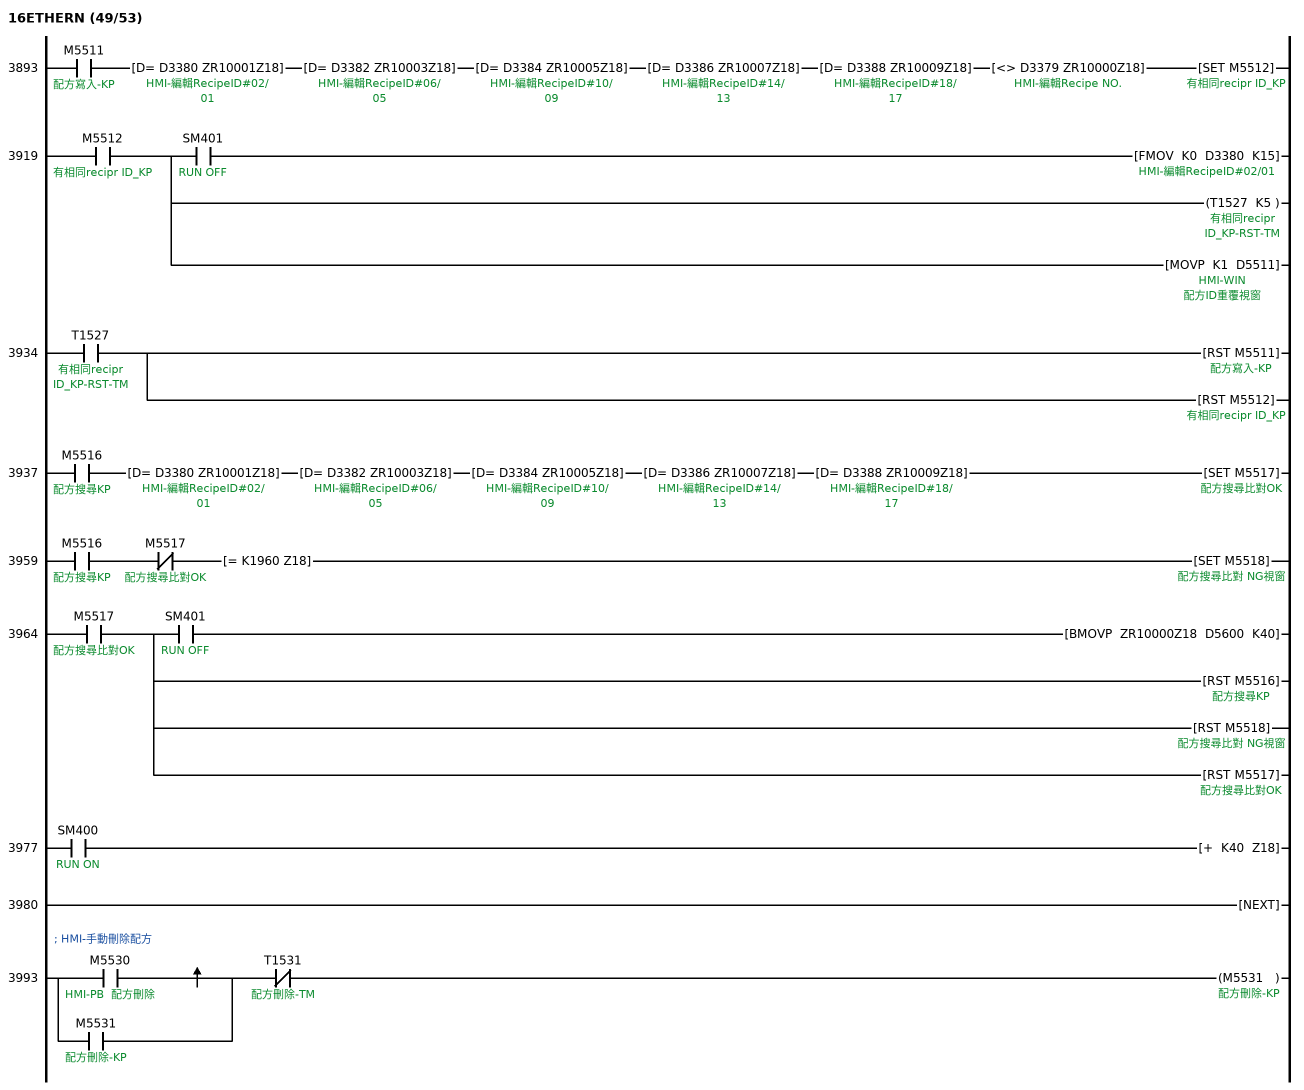
3893  LD      M5511  ; 配方寫入-KP
      ANDD=   D3380 ZR10001Z18  ; HMI-編輯RecipeID#02/01
      ANDD=   D3382 ZR10003Z18  ; HMI-編輯RecipeID#06/05
      ANDD=   D3384 ZR10005Z18  ; HMI-編輯RecipeID#10/09
      ANDD=   D3386 ZR10007Z18  ; HMI-編輯RecipeID#14/13
      ANDD=   D3388 ZR10009Z18  ; HMI-編輯RecipeID#18/17
      AND<>   D3379 ZR10000Z18  ; HMI-編輯Recipe NO.
      SET     M5512  ; 有相同recipr ID_KP
3919  LD      M5512  ; 有相同recipr ID_KP
      MPS
      AND     SM401  ; RUN OFF
      FMOV    K0 D3380 K15
      MPP
      OUT     T1527 K5  ; 有相同recipr ID_KP-RST-TM
      MOVP    K1 D5511
3934  LD      T1527  ; 有相同recipr ID_KP-RST-TM
      RST     M5511  ; 配方寫入-KP
      RST     M5512  ; 有相同recipr ID_KP
3937  LD      M5516  ; 配方搜尋KP
      ANDD=   D3380 ZR10001Z18  ; HMI-編輯RecipeID#02/01
      ANDD=   D3382 ZR10003Z18  ; HMI-編輯RecipeID#06/05
      ANDD=   D3384 ZR10005Z18  ; HMI-編輯RecipeID#10/09
      ANDD=   D3386 ZR10007Z18  ; HMI-編輯RecipeID#14/13
      ANDD=   D3388 ZR10009Z18  ; HMI-編輯RecipeID#18/17
      SET     M5517  ; 配方搜尋比對OK
3959  LD      M5516  ; 配方搜尋KP
      ANI     M5517  ; 配方搜尋比對OK
      AND=    K1960 Z18
      SET     M5518  ; 配方搜尋比對 NG視窗
3964  LD      M5517  ; 配方搜尋比對OK
      MPS
      AND     SM401  ; RUN OFF
      BMOVP   ZR10000Z18 D5600 K40
      MPP
      RST     M5516  ; 配方搜尋KP
      RST     M5518  ; 配方搜尋比對 NG視窗
      RST     M5517  ; 配方搜尋比對OK
3977  LD      SM400  ; RUN ON
      +       K40 Z18
3980  NEXT
; HMI-手動刪除配方
3993  LD      M5530  ; HMI-PB  配方刪除
      MEP
      OR      M5531  ; 配方刪除-KP
      ANI     T1531  ; 配方刪除-TM
      OUT     M5531  ; 配方刪除-KP
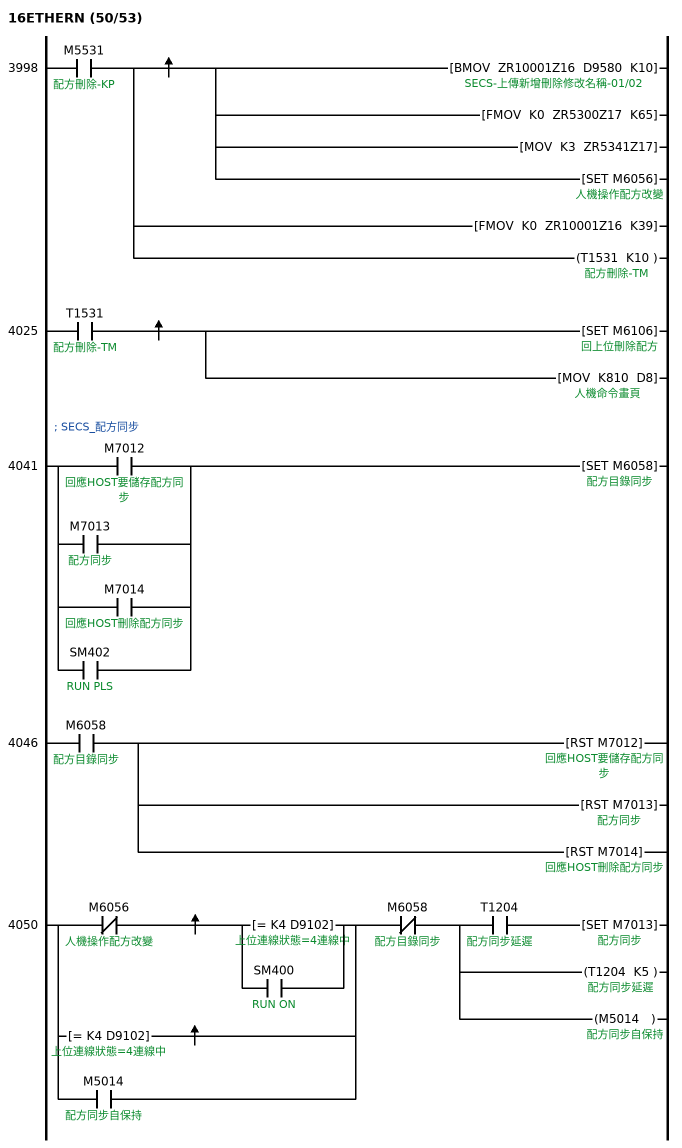
3998  LD      M5531  ; 配方刪除-KP
      MPS
      MEP
      BMOV    ZR10001Z16 D9580 K10
      FMOV    K0 ZR5300Z17 K65
      MOV     K3 ZR5341Z17
      SET     M6056  ; 人機操作配方改變
      MPP
      FMOV    K0 ZR10001Z16 K39
      OUT     T1531 K10  ; 配方刪除-TM
4025  LD      T1531  ; 配方刪除-TM
      MEP
      SET     M6106  ; 回上位刪除配方
      MOV     K810 D8
; SECS_配方同步
4041  LD      M7012  ; 回應HOST要儲存配方同步
      OR      M7013  ; 配方同步
      OR      M7014  ; 回應HOST刪除配方同步
      OR      SM402  ; RUN PLS
      SET     M6058  ; 配方目錄同步
4046  LD      M6058  ; 配方目錄同步
      RST     M7012  ; 回應HOST要儲存配方同步
      RST     M7013  ; 配方同步
      RST     M7014  ; 回應HOST刪除配方同步
4050  LDI     M6056  ; 人機操作配方改變
      MEP
      LD=     K4 D9102  ; 上位連線狀態=4連線中
      OR      SM400  ; RUN ON
      ANB
      LD=     K4 D9102  ; 上位連線狀態=4連線中
      MEP
      ORB
      OR      M5014  ; 配方同步自保持
      ANI     M6058  ; 配方目錄同步
      MPS
      AND     T1204  ; 配方同步延遲
      SET     M7013  ; 配方同步
      MPP
      OUT     T1204 K5  ; 配方同步延遲
      OUT     M5014  ; 配方同步自保持
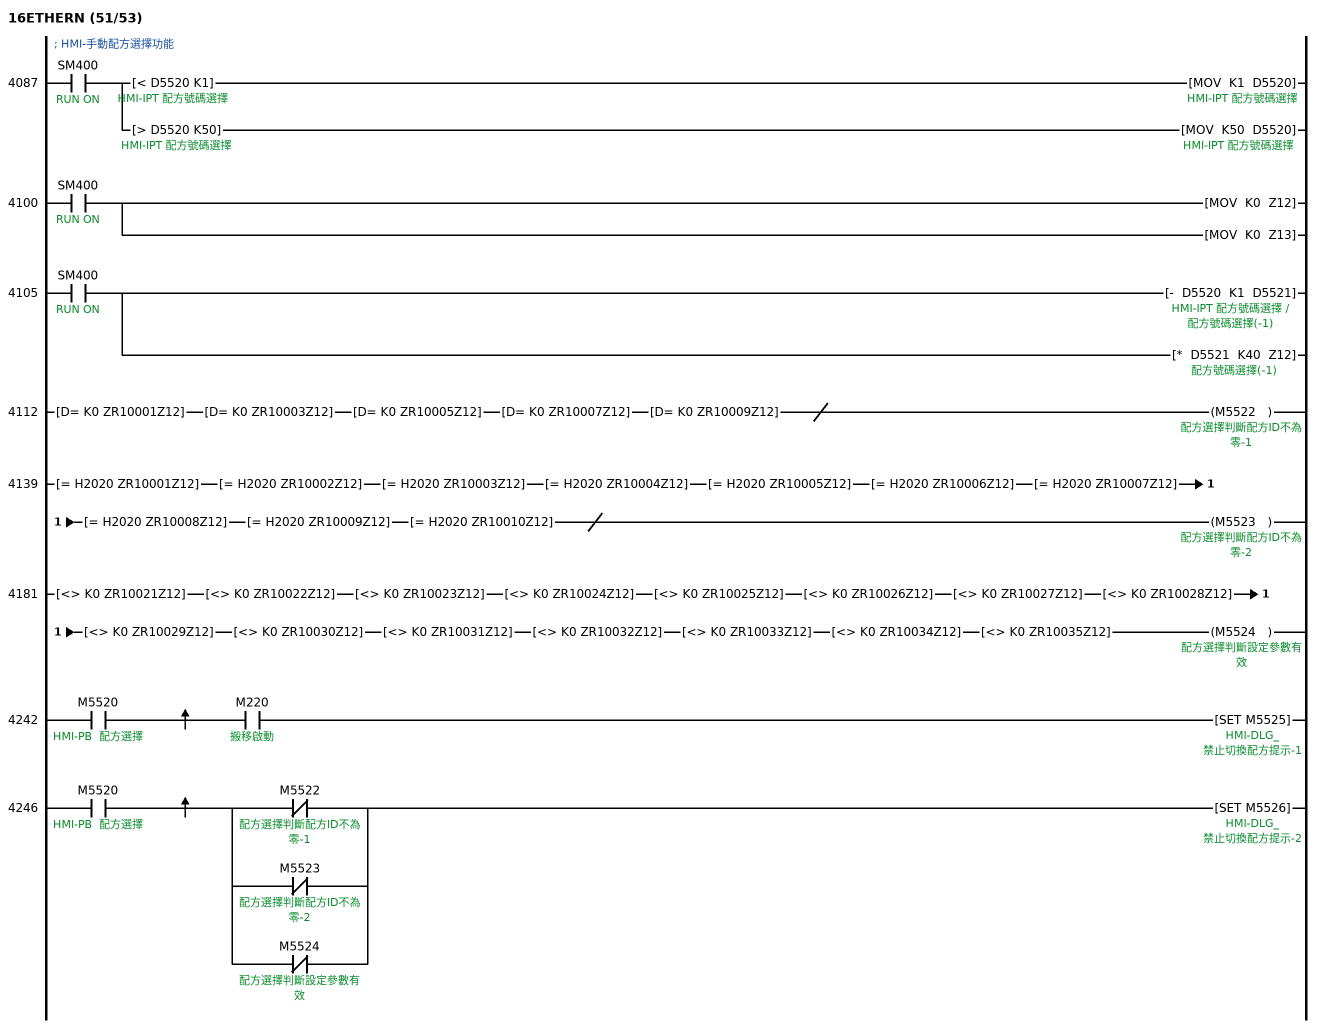
; HMI-手動配方選擇功能
4087  LD      SM400  ; RUN ON
      MPS
      AND<    D5520 K1  ; HMI-IPT 配方號碼選擇
      MOV     K1 D5520
      MPP
      AND>    D5520 K50  ; HMI-IPT 配方號碼選擇
      MOV     K50 D5520
4100  LD      SM400  ; RUN ON
      MOV     K0 Z12
      MOV     K0 Z13
4105  LD      SM400  ; RUN ON
      -       D5520 K1 D5521  ; 配方號碼選擇(-1)
      *       D5521 K40 Z12
4112  LDD=    K0 ZR10001Z12
      ANDD=   K0 ZR10003Z12
      ANDD=   K0 ZR10005Z12
      ANDD=   K0 ZR10007Z12
      ANDD=   K0 ZR10009Z12
      INV
      OUT     M5522  ; 配方選擇判斷配方ID不為零-1
4139  LD=     H2020 ZR10001Z12
      AND=    H2020 ZR10002Z12
      AND=    H2020 ZR10003Z12
      AND=    H2020 ZR10004Z12
      AND=    H2020 ZR10005Z12
      AND=    H2020 ZR10006Z12
      AND=    H2020 ZR10007Z12
      AND=    H2020 ZR10008Z12
      AND=    H2020 ZR10009Z12
      AND=    H2020 ZR10010Z12
      INV
      OUT     M5523  ; 配方選擇判斷配方ID不為零-2
4181  LD<>    K0 ZR10021Z12
      AND<>   K0 ZR10022Z12
      AND<>   K0 ZR10023Z12
      AND<>   K0 ZR10024Z12
      AND<>   K0 ZR10025Z12
      AND<>   K0 ZR10026Z12
      AND<>   K0 ZR10027Z12
      AND<>   K0 ZR10028Z12
      AND<>   K0 ZR10029Z12
      AND<>   K0 ZR10030Z12
      AND<>   K0 ZR10031Z12
      AND<>   K0 ZR10032Z12
      AND<>   K0 ZR10033Z12
      AND<>   K0 ZR10034Z12
      AND<>   K0 ZR10035Z12
      OUT     M5524  ; 配方選擇判斷設定參數有效
4242  LD      M5520  ; HMI-PB  配方選擇
      MEP
      AND     M220  ; 搬移啟動
      SET     M5525  ; HMI-DLG_禁止切換配方提示-1
4246  LD      M5520  ; HMI-PB  配方選擇
      MEP
      LDI     M5522  ; 配方選擇判斷配方ID不為零-1
      ORI     M5523  ; 配方選擇判斷配方ID不為零-2
      ORI     M5524  ; 配方選擇判斷設定參數有效
      ANB
      SET     M5526  ; HMI-DLG_禁止切換配方提示-2
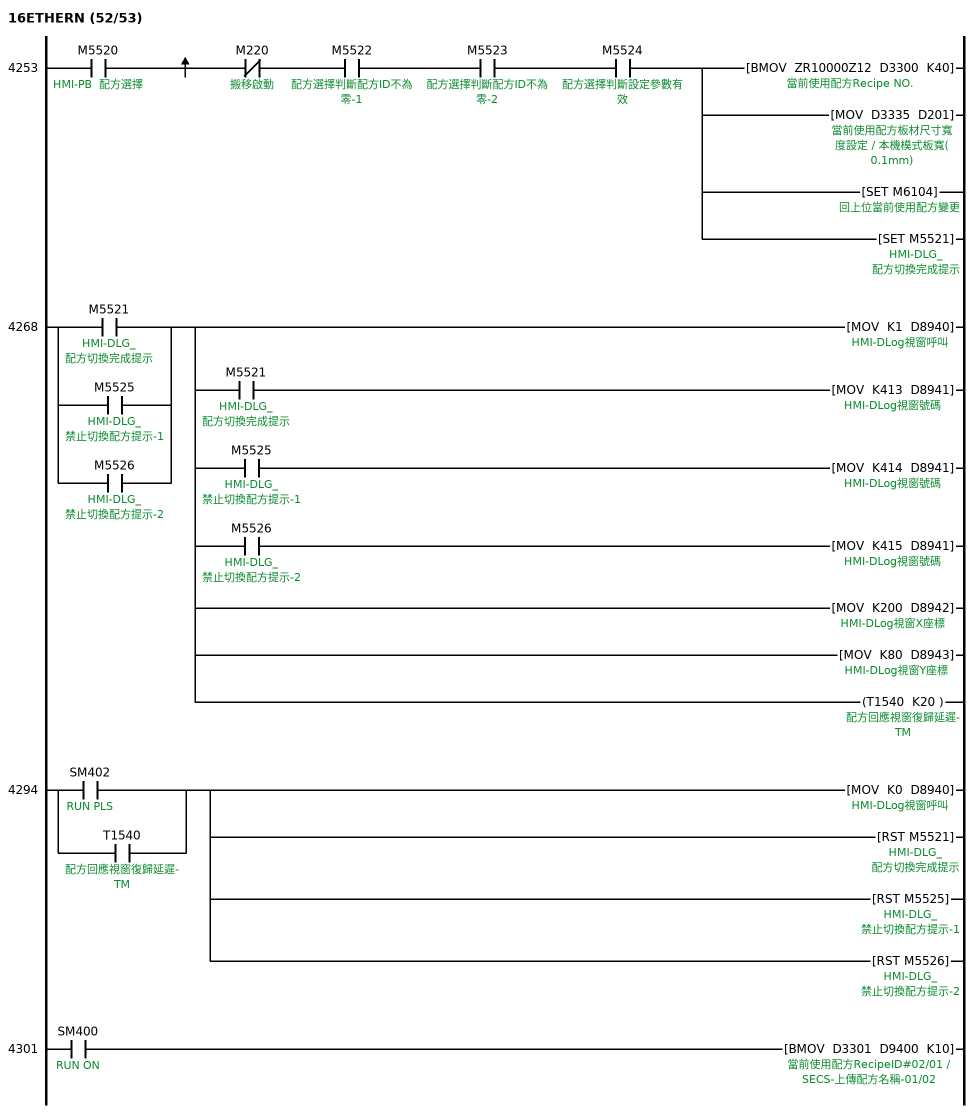
4253  LD      M5520  ; HMI-PB  配方選擇
      MEP
      ANI     M220  ; 搬移啟動
      AND     M5522  ; 配方選擇判斷配方ID不為零-1
      AND     M5523  ; 配方選擇判斷配方ID不為零-2
      AND     M5524  ; 配方選擇判斷設定參數有效
      BMOV    ZR10000Z12 D3300 K40
      MOV     D3335 D201
      SET     M6104  ; 回上位當前使用配方變更
      SET     M5521  ; HMI-DLG_配方切換完成提示
4268  LD      M5521  ; HMI-DLG_配方切換完成提示
      OR      M5525  ; HMI-DLG_禁止切換配方提示-1
      OR      M5526  ; HMI-DLG_禁止切換配方提示-2
      MOV     K1 D8940  ; HMI-DLog視窗呼叫
      MPS
      AND     M5521  ; HMI-DLG_配方切換完成提示
      MOV     K413 D8941  ; HMI-DLog視窗號碼
      MRD
      AND     M5525  ; HMI-DLG_禁止切換配方提示-1
      MOV     K414 D8941
      MRD
      AND     M5526  ; HMI-DLG_禁止切換配方提示-2
      MOV     K415 D8941
      MPP
      MOV     K200 D8942  ; HMI-DLog視窗X座標
      MOV     K80 D8943  ; HMI-DLog視窗Y座標
      OUT     T1540 K20  ; 配方回應視窗復歸延遲-TM
4294  LD      SM402  ; RUN PLS
      OR      T1540  ; 配方回應視窗復歸延遲-TM
      MOV     K0 D8940
      RST     M5521  ; HMI-DLG_配方切換完成提示
      RST     M5525  ; HMI-DLG_禁止切換配方提示-1
      RST     M5526  ; HMI-DLG_禁止切換配方提示-2
4301  LD      SM400  ; RUN ON
      BMOV    D3301 D9400 K10  ; 當前使用配方RecipeID#02/01 / SECS-上傳配方名稱-01/02
        [note] D9400_上報SECS目前使用PPID名稱
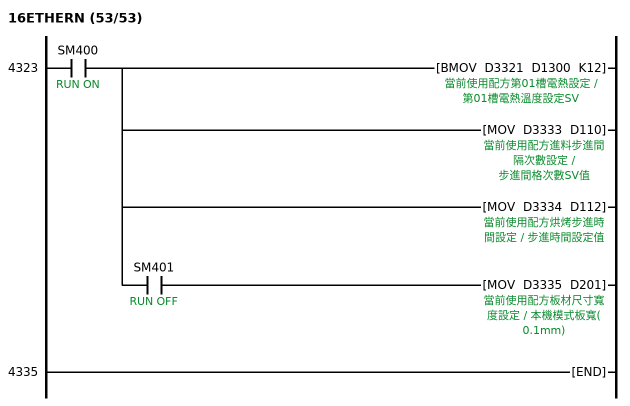
4323  LD      SM400  ; RUN ON
      BMOV    D3321 D1300 K12  ; 當前使用配方第01槽電熱設定
      MOV     D3333 D110  ; 當前使用配方進料步進間隔次數設定
      MOV     D3334 D112  ; 當前使用配方烘烤步進時間設定
      AND     SM401  ; RUN OFF
      MOV     D3335 D201
4335  END
END_PROGRAM

PROGRAM 17GBF-20
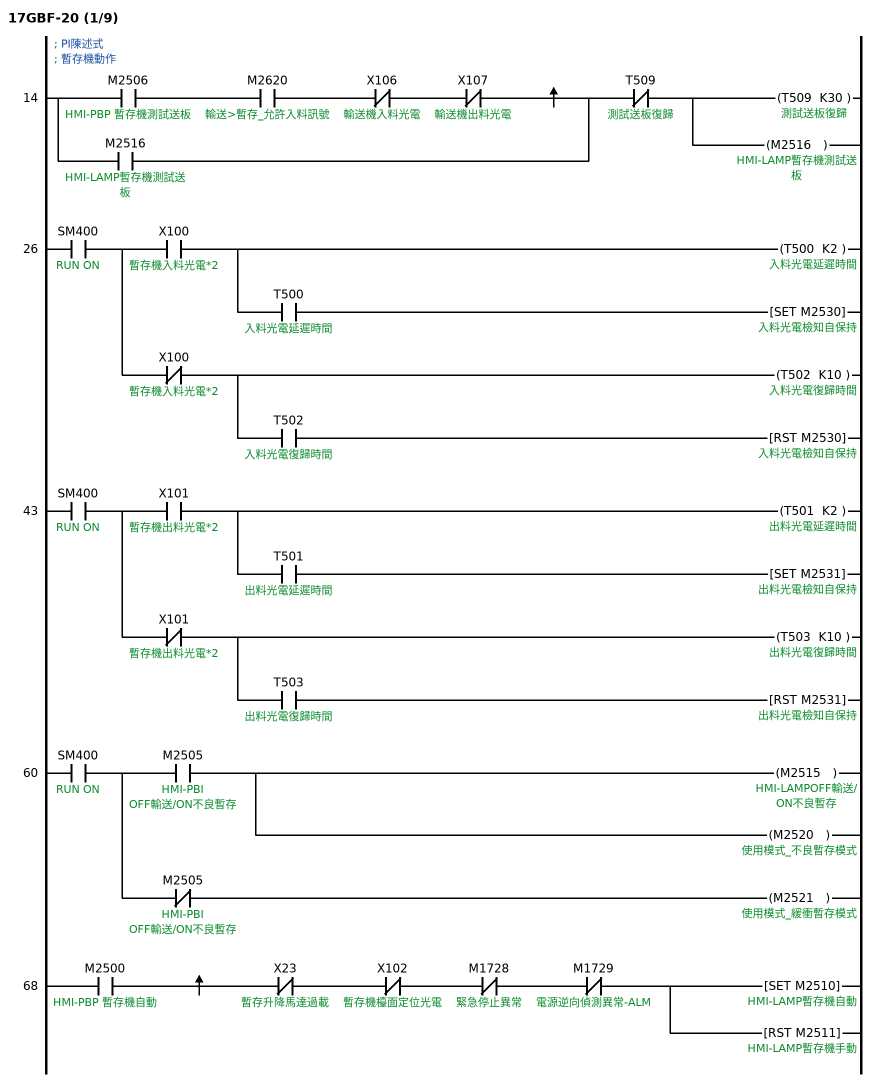
; PI陳述式
; 暫存機動作
14    LD      M2506  ; HMI-PBP 暫存機測試送板
      AND     M2620  ; 輸送>暫存_允許入料訊號
      ANI     X106  ; 輸送機入料光電
      ANI     X107  ; 輸送機出料光電
      MEP
      OR      M2516  ; HMI-LAMP暫存機測試送板
      ANI     T509  ; 測試送板復歸
      OUT     T509 K30  ; 測試送板復歸
      OUT     M2516  ; HMI-LAMP暫存機測試送板
26    LD      SM400  ; RUN ON
      MPS
      AND     X100  ; 暫存機入料光電*2
      OUT     T500 K2  ; 入料光電延遲時間
      AND     T500  ; 入料光電延遲時間
      SET     M2530  ; 入料光電檢知自保持
      MPP
      ANI     X100  ; 暫存機入料光電*2
      OUT     T502 K10  ; 入料光電復歸時間
      AND     T502  ; 入料光電復歸時間
      RST     M2530  ; 入料光電檢知自保持
43    LD      SM400  ; RUN ON
      MPS
      AND     X101  ; 暫存機出料光電*2
      OUT     T501 K2  ; 出料光電延遲時間
      AND     T501  ; 出料光電延遲時間
      SET     M2531  ; 出料光電檢知自保持
      MPP
      ANI     X101  ; 暫存機出料光電*2
      OUT     T503 K10  ; 出料光電復歸時間
      AND     T503  ; 出料光電復歸時間
      RST     M2531  ; 出料光電檢知自保持
60    LD      SM400  ; RUN ON
      MPS
      AND     M2505  ; HMI-PBI OFF輸送/ON不良暫存
      OUT     M2515  ; HMI-LAMPOFF輸送/ON不良暫存
      OUT     M2520  ; 使用模式_不良暫存模式
      MPP
      ANI     M2505  ; HMI-PBI OFF輸送/ON不良暫存
      OUT     M2521  ; 使用模式_緩衝暫存模式
68    LD      M2500  ; HMI-PBP 暫存機自動
      MEP
      ANI     X23  ; 暫存升降馬達過載
      ANI     X102  ; 暫存機檯面定位光電
      ANI     M1728  ; 緊急停止異常
      ANI     M1729  ; 電源逆向偵測異常-ALM
      SET     M2510  ; HMI-LAMP暫存機自動
      RST     M2511  ; HMI-LAMP暫存機手動
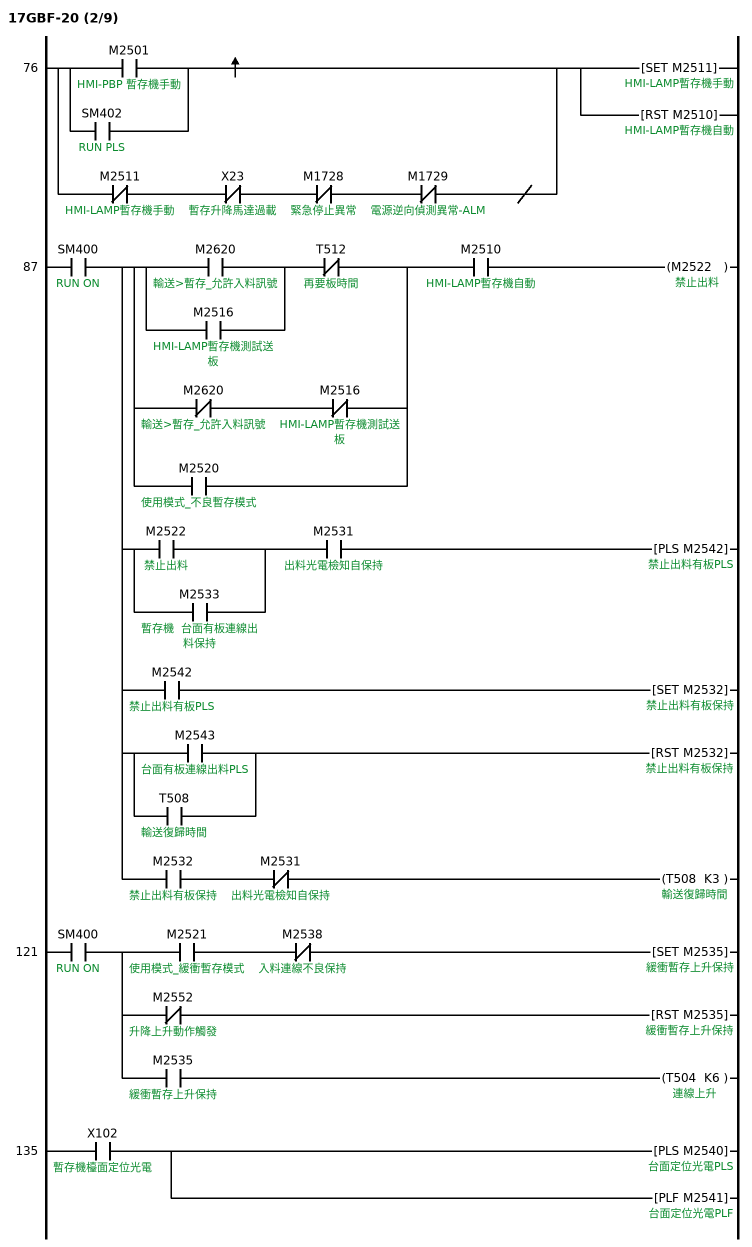
76    LD      M2501  ; HMI-PBP 暫存機手動
      OR      SM402  ; RUN PLS
      MEP
      LDI     M2511  ; HMI-LAMP暫存機手動
      ANI     X23  ; 暫存升降馬達過載
      ANI     M1728  ; 緊急停止異常
      ANI     M1729  ; 電源逆向偵測異常-ALM
      INV
      ORB
      SET     M2511  ; HMI-LAMP暫存機手動
      RST     M2510  ; HMI-LAMP暫存機自動
87    LD      SM400  ; RUN ON
      MPS
      LD      M2620  ; 輸送>暫存_允許入料訊號
      OR      M2516  ; HMI-LAMP暫存機測試送板
      ANI     T512  ; 再要板時間
      LDI     M2620  ; 輸送>暫存_允許入料訊號
      ANI     M2516  ; HMI-LAMP暫存機測試送板
      ORB
      OR      M2520  ; 使用模式_不良暫存模式
      ANB
      AND     M2510  ; HMI-LAMP暫存機自動
      OUT     M2522  ; 禁止出料
      MRD
      LD      M2522  ; 禁止出料
      OR      M2533  ; 暫存機  台面有板連線出料保持
      ANB
      AND     M2531  ; 出料光電檢知自保持
      PLS     M2542  ; 禁止出料有板PLS
      MRD
      AND     M2542  ; 禁止出料有板PLS
      SET     M2532  ; 禁止出料有板保持
      MRD
      LD      M2543  ; 台面有板連線出料PLS
      OR      T508  ; 輸送復歸時間
      ANB
      RST     M2532  ; 禁止出料有板保持
      MPP
      AND     M2532  ; 禁止出料有板保持
      ANI     M2531  ; 出料光電檢知自保持
      OUT     T508 K3  ; 輸送復歸時間
121   LD      SM400  ; RUN ON
      MPS
      AND     M2521  ; 使用模式_緩衝暫存模式
      ANI     M2538  ; 入料連線不良保持
      SET     M2535  ; 緩衝暫存上升保持
      MRD
      ANI     M2552  ; 升降上升動作觸發
      RST     M2535  ; 緩衝暫存上升保持
      MPP
      AND     M2535  ; 緩衝暫存上升保持
      OUT     T504 K6  ; 連線上升
135   LD      X102  ; 暫存機檯面定位光電
      PLS     M2540  ; 台面定位光電PLS
      PLF     M2541  ; 台面定位光電PLF
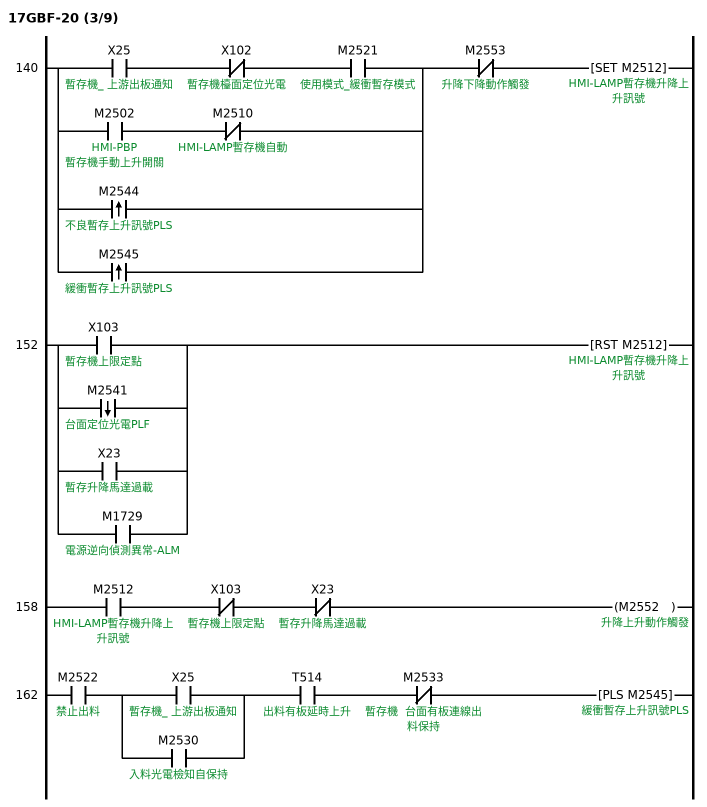
140   LD      X25  ; 暫存機_ 上游出板通知
      ANI     X102  ; 暫存機檯面定位光電
      AND     M2521  ; 使用模式_緩衝暫存模式
      LD      M2502  ; HMI-PBP 暫存機手動上升開關
      ANI     M2510  ; HMI-LAMP暫存機自動
      ORB
      ORP     M2544  ; 不良暫存上升訊號PLS
      ORP     M2545  ; 緩衝暫存上升訊號PLS
      ANI     M2553  ; 升降下降動作觸發
      SET     M2512  ; HMI-LAMP暫存機升降上升訊號
152   LD      X103  ; 暫存機上限定點
      ORF     M2541  ; 台面定位光電PLF
      OR      X23  ; 暫存升降馬達過載
      OR      M1729  ; 電源逆向偵測異常-ALM
      RST     M2512  ; HMI-LAMP暫存機升降上升訊號
158   LD      M2512  ; HMI-LAMP暫存機升降上升訊號
      ANI     X103  ; 暫存機上限定點
      ANI     X23  ; 暫存升降馬達過載
      OUT     M2552  ; 升降上升動作觸發
162   LD      M2522  ; 禁止出料
      LD      X25  ; 暫存機_ 上游出板通知
      OR      M2530  ; 入料光電檢知自保持
      ANB
      AND     T514  ; 出料有板延時上升
      ANI     M2533  ; 暫存機  台面有板連線出料保持
      PLS     M2545  ; 緩衝暫存上升訊號PLS
